LIN {X 0,Y 336.129,Z 1041.113,A -85,B 0,C 180,E1 25405.628,E2 25405.628} C_VEL
LIN {X 0,Y 318.672,Z 1080.117,A -85,B 0,C 180,E1 25408.835,E2 25408.835} C_VEL
LIN {X 0,Y 298.795,Z 1116.073,A -85,B 0,C 180,E1 25413.198,E2 25413.198} C_VEL
LIN {X 0,Y 277.626,Z 1148.443,A -85,B 0,C 180,E1 25419.027,E2 25419.027} C_VEL
LIN {X 0,Y 257.542,Z 1176.137,A -85,B 0,C 180,E1 25426.627,E2 25426.627} C_VEL
LIN {X 0,Y 241.568,Z 1197.526,A -85,B 0,C 180,E1 25435.629,E2 25435.629} C_VEL
LIN {X 0,Y 230.931,Z 1212.917,A -85,B 0,C 180,E1 25445.788,E2 25445.788} C_VEL
LIN {X 0,Y 226.21,Z 1222.177,A -85,B 0,C 180,E1 25455.992,E2 25455.992} C_VEL
LIN {X 0,Y 224.98,Z 1226.535,A -85,B 0,C 180,E1 25466.138,E2 25466.138} C_VEL
LIN {X 0,Y 225.27,Z 1226.905,A -85,B 0,C 180,E1 25470,E2 25470} C_VEL
LIN {X 0,Y 225.086,Z 1225.472,A -85,B 0,C 180,E1 25477.737,E2 25477.737} C_VEL
LIN {X 0,Y 227.29,Z 1219.666,A -85,B 0,C 180,E1 25487.457,E2 25487.457} C_VEL
LIN {X 0,Y 234.034,Z 1208.265,A -85,B 0,C 180,E1 25497.865,E2 25497.865} C_VEL
LIN {X 0,Y 246.932,Z 1190.434,A -85,B 0,C 180,E1 25507.853,E2 25507.853} C_VEL
LIN {X 0,Y 265.132,Z 1166.006,A -85,B 0,C 180,E1 25516.595,E2 25516.595} C_VEL
LIN {X 0,Y 285.468,Z 1137.166,A -85,B 0,C 180,E1 25523.324,E2 25523.324} C_VEL
LIN {X 0,Y 306.843,Z 1102.563,A -85,B 0,C 180,E1 25528.679,E2 25528.679} C_VEL
LIN {X 0,Y 326.303,Z 1064.734,A -85,B 0,C 180,E1 25532.594,E2 25532.594} C_VEL
LIN {X 0,Y 336.503,Z 1040.269,A -85,B 0,C 180,E1 25534.514,E2 25534.514} C_VEL
LIN {X 0,Y 333.813,Z 1018.325,A -85,B 0,C 180,E1 25539.751,E2 25539.751} C_VEL
LIN {X 0,Y 329.876,Z 1000.5,A -85,B 0,C 180,E1 25545.365,E2 25545.365} C_VEL
LIN {X 0,Y 326.385,Z 988.649,A -85,B 0,C 180,E1 25550.647,E2 25550.647} C_VEL
LIN {X 0,Y 324.003,Z 980.521,A -85,B 0,C 180,E1 25556.143,E2 25556.143} C_VEL
LIN {X 0,Y 323.437,Z 975.758,A -85,B 0,C 180,E1 25561.338,E2 25561.338} C_VEL
LIN {X 0,Y 323.425,Z 976.928,A -85,B 0,C 180,E1 25565.372,E2 25565.372} C_VEL
LIN {X 0,Y 325.459,Z 983.529,A -85,B 0,C 180,E1 25571.883,E2 25571.883} C_VEL
LIN {X 0,Y 329.595,Z 994.792,A -85,B 0,C 180,E1 25578.07,E2 25578.07} C_VEL
LIN {X 0,Y 334.739,Z 1011.693,A -85,B 0,C 180,E1 25584.032,E2 25584.032} C_VEL
LIN {X 0,Y 339.138,Z 1032.622,A -85,B 0,C 180,E1 25589.426,E2 25589.426} C_VEL
LIN {X 0,Y 339.403,Z 1039.091,A -85,B 0,C 180,E1 25590.675,E2 25590.675} C_VEL
LIN {X 0,Y 333.764,Z 1052.968,A -85,B 0,C 180,E1 25591.555,E2 25591.555} C_VEL
LIN {X 0,Y 325.121,Z 1067.998,A -85,B 0,C 180,E1 25592.055,E2 25592.055} C_VEL
LIN {X 0,Y 315.788,Z 1082.353,A -85,B 0,C 180,E1 25592.714,E2 25592.714} C_VEL
LIN {X 0,Y 295.451,Z 1116.69,A -85,B 0,C 180,E1 25596.74,E2 25596.74} C_VEL
LIN {X 0,Y 274.846,Z 1145.734,A -85,B 0,C 180,E1 25601.903,E2 25601.903} C_VEL
LIN {X 0,Y 255.367,Z 1169.768,A -85,B 0,C 180,E1 25608.418,E2 25608.418} C_VEL
LIN {X 0,Y 237.524,Z 1190.148,A -85,B 0,C 180,E1 25617.163,E2 25617.163} C_VEL
LIN {X 0,Y 225.183,Z 1204.304,A -85,B 0,C 180,E1 25627.237,E2 25627.237} C_VEL
LIN {X 0,Y 218.796,Z 1212.593,A -85,B 0,C 180,E1 25638.009,E2 25638.009} C_VEL
LIN {X 0,Y 217.331,Z 1215.277,A -85,B 0,C 180,E1 25646.002,E2 25646.002} C_VEL
LIN {X 0,Y 217.346,Z 1215.244,A -85,B 0,C 180,E1 25653.998,E2 25653.998} C_VEL
LIN {X 0,Y 219.664,Z 1211.343,A -85,B 0,C 180,E1 25663.972,E2 25663.972} C_VEL
LIN {X 0,Y 226.955,Z 1202.026,A -85,B 0,C 180,E1 25674.593,E2 25674.593} C_VEL
LIN {X 0,Y 239.047,Z 1188.251,A -85,B 0,C 180,E1 25683.687,E2 25683.687} C_VEL
LIN {X 0,Y 255.629,Z 1169.328,A -85,B 0,C 180,E1 25691.581,E2 25691.581} C_VEL
LIN {X 0,Y 276.15,Z 1143.785,A -85,B 0,C 180,E1 25698.386,E2 25698.386} C_VEL
LIN {X 0,Y 297.513,Z 1113.138,A -85,B 0,C 180,E1 25703.646,E2 25703.646} C_VEL
LIN {X 0,Y 316.98,Z 1079.695,A -85,B 0,C 180,E1 25707.411,E2 25707.411} C_VEL
LIN {X 0,Y 334.005,Z 1042.885,A -85,B 0,C 180,E1 25710.188,E2 25710.188} C_VEL
LIN {X 0,Y 334.535,Z 1040.217,A -85,B 0,C 180,E1 25710.507,E2 25710.507} C_VEL
LIN {X 0,Y 331.211,Z 1019.932,A -85,B 0,C 180,E1 25715.696,E2 25715.696} C_VEL
LIN {X 0,Y 327.07,Z 1004.267,A -85,B 0,C 180,E1 25721.086,E2 25721.086} C_VEL
LIN {X 0,Y 323.534,Z 993.29,A -85,B 0,C 180,E1 25726.464,E2 25726.464} C_VEL
LIN {X 0,Y 321.586,Z 987.722,A -85,B 0,C 180,E1 25730.856,E2 25730.856} C_VEL
LIN {X 0,Y 320.944,Z 983.41,A -85,B 0,C 180,E1 25735.608,E2 25735.608} C_VEL
LIN {X 0,Y 320.957,Z 983.923,A -85,B 0,C 180,E1 25740.004,E2 25740.004} C_VEL
LIN {X 0,Y 322.266,Z 991.69,A -85,B 0,C 180,E1 25746.753,E2 25746.753} C_VEL
LIN {X 0,Y 325.363,Z 1003.281,A -85,B 0,C 180,E1 25752.78,E2 25752.78} C_VEL
LIN {X 0,Y 328.73,Z 1019.789,A -85,B 0,C 180,E1 25758.475,E2 25758.475} C_VEL
LIN {X 0,Y 330.979,Z 1038.496,A -85,B 0,C 180,E1 25763.34,E2 25763.34} C_VEL
LIN {X 0,Y 331.241,Z 1043.446,A -85,B 0,C 180,E1 25764.489,E2 25764.489} C_VEL
LIN {X 0,Y 314.299,Z 1080.693,A -85,B 0,C 180,E1 25767.642,E2 25767.642} C_VEL
LIN {X 0,Y 294.401,Z 1115.737,A -85,B 0,C 180,E1 25771.868,E2 25771.868} C_VEL
LIN {X 0,Y 272.508,Z 1148.223,A -85,B 0,C 180,E1 25777.703,E2 25777.703} C_VEL
LIN {X 0,Y 252.237,Z 1175.168,A -85,B 0,C 180,E1 25785.089,E2 25785.089} C_VEL
LIN {X 0,Y 234.855,Z 1197.301,A -85,B 0,C 180,E1 25794.501,E2 25794.501} C_VEL
LIN {X 0,Y 223.565,Z 1212.701,A -85,B 0,C 180,E1 25804.936,E2 25804.936} C_VEL
LIN {X 0,Y 218.869,Z 1220.981,A -85,B 0,C 180,E1 25813.922,E2 25813.922} C_VEL
LIN {X 0,Y 217.198,Z 1225.254,A -85,B 0,C 180,E1 25821.979,E2 25821.979} C_VEL
LIN {X 0,Y 217.362,Z 1226.703,A -85,B 0,C 180,E1 25829.999,E2 25829.999} C_VEL
LIN {X 0,Y 217.194,Z 1225.269,A -85,B 0,C 180,E1 25838.02,E2 25838.02} C_VEL
LIN {X 0,Y 219.606,Z 1219.459,A -85,B 0,C 180,E1 25848.089,E2 25848.089} C_VEL
LIN {X 0,Y 227.281,Z 1207.429,A -85,B 0,C 180,E1 25859.253,E2 25859.253} C_VEL
LIN {X 0,Y 241.219,Z 1189.193,A -85,B 0,C 180,E1 25869.496,E2 25869.496} C_VEL
LIN {X 0,Y 259.567,Z 1165.746,A -85,B 0,C 180,E1 25877.91,E2 25877.91} C_VEL
LIN {X 0,Y 280.555,Z 1137.014,A -85,B 0,C 180,E1 25884.636,E2 25884.636} C_VEL
LIN {X 0,Y 302.436,Z 1102.655,A -85,B 0,C 180,E1 25889.936,E2 25889.936} C_VEL
LIN {X 0,Y 322.305,Z 1065.017,A -85,B 0,C 180,E1 25893.804,E2 25893.804} C_VEL
LIN {X 0,Y 331.473,Z 1043.453,A -85,B 0,C 180,E1 25895.529,E2 25895.529} C_VEL
LIN {X 0,Y 329.352,Z 1022.205,A -85,B 0,C 180,E1 25900.866,E2 25900.866} C_VEL
LIN {X 0,Y 325.746,Z 1004.055,A -85,B 0,C 180,E1 25906.979,E2 25906.979} C_VEL
LIN {X 0,Y 323.126,Z 993.991,A -85,B 0,C 180,E1 25911.911,E2 25911.911} C_VEL
LIN {X 0,Y 321.841,Z 988.466,A -85,B 0,C 180,E1 25915.61,E2 25915.61} C_VEL
LIN {X 0,Y 321.245,Z 983.354,A -85,B 0,C 180,E1 25921.347,E2 25921.347} C_VEL
LIN {X 0,Y 321.208,Z 984.556,A -85,B 0,C 180,E1 25925.301,E2 25925.301} C_VEL
LIN {X 0,Y 323.21,Z 991.921,A -85,B 0,C 180,E1 25932.356,E2 25932.356} C_VEL
LIN {X 0,Y 326.909,Z 1003.008,A -85,B 0,C 180,E1 25938.224,E2 25938.224} C_VEL
LIN {X 0,Y 331.466,Z 1020.386,A -85,B 0,C 180,E1 25944.284,E2 25944.284} C_VEL
LIN {X 0,Y 334.788,Z 1040.967,A -85,B 0,C 180,E1 25949.529,E2 25949.529} C_VEL
LIN {X 0,Y 317.498,Z 1079.101,A -85,B 0,C 180,E1 25952.419,E2 25952.419} C_VEL
LIN {X 0,Y 315.788,Z 1082.353,A -85,B 0,C 180,E1 25952.714,E2 25952.714} C_VEL
LIN {X 0,Y 305.838,Z 1096.298,A -85,B 0,C 180,E1 25953.5,E2 25953.5} C_VEL
LIN {X 0,Y 295.657,Z 1109.492,A -85,B 0,C 180,E1 25954.46,E2 25954.46} C_VEL
LIN {X 0,Y 275.018,Z 1138.959,A -85,B 0,C 180,E1 25959.196,E2 25959.196} C_VEL
LIN {X 0,Y 254.976,Z 1163.672,A -85,B 0,C 180,E1 25965.197,E2 25965.197} C_VEL
LIN {X 0,Y 235.982,Z 1184.766,A -85,B 0,C 180,E1 25973.177,E2 25973.177} C_VEL
LIN {X 0,Y 221.688,Z 1200.233,A -85,B 0,C 180,E1 25982.654,E2 25982.654} C_VEL
LIN {X 0,Y 212.851,Z 1210.407,A -85,B 0,C 180,E1 25993.456,E2 25993.456} C_VEL
LIN {X 0,Y 209.89,Z 1214.484,A -85,B 0,C 180,E1 26001.699,E2 26001.699} C_VEL
LIN {X 0,Y 209.529,Z 1215.793,A -85,B 0,C 180,E1 26010.001,E2 26010.001} C_VEL
LIN {X 0,Y 209.925,Z 1214.421,A -85,B 0,C 180,E1 26018.301,E2 26018.301} C_VEL
LIN {X 0,Y 214.055,Z 1208.79,A -85,B 0,C 180,E1 26028.576,E2 26028.576} C_VEL
LIN {X 0,Y 224.162,Z 1197.308,A -85,B 0,C 180,E1 26039.347,E2 26039.347} C_VEL
LIN {X 0,Y 239.611,Z 1180.675,A -85,B 0,C 180,E1 26048.524,E2 26048.524} C_VEL
LIN {X 0,Y 258.431,Z 1159.363,A -85,B 0,C 180,E1 26055.913,E2 26055.913} C_VEL
LIN {X 0,Y 279.416,Z 1132.799,A -85,B 0,C 180,E1 26061.846,E2 26061.846} C_VEL
LIN {X 0,Y 300.375,Z 1101.648,A -85,B 0,C 180,E1 26066.403,E2 26066.403} C_VEL
LIN {X 0,Y 319.816,Z 1066.366,A -85,B 0,C 180,E1 26069.79,E2 26069.79} C_VEL
LIN {X 0,Y 329.382,Z 1045.22,A -85,B 0,C 180,E1 26071.277,E2 26071.277} C_VEL
LIN {X 0,Y 327.702,Z 1028.663,A -85,B 0,C 180,E1 26075.419,E2 26075.419} C_VEL
LIN {X 0,Y 324.087,Z 1012.395,A -85,B 0,C 180,E1 26080.905,E2 26080.905} C_VEL
LIN {X 0,Y 320.969,Z 1001.103,A -85,B 0,C 180,E1 26086.354,E2 26086.354} C_VEL
LIN {X 0,Y 318.634,Z 994,A -85,B 0,C 180,E1 26092.266,E2 26092.266} C_VEL
LIN {X 0,Y 318.522,Z 991.648,A -85,B 0,C 180,E1 26094.546,E2 26094.546} C_VEL
LIN {X 0,Y 318.408,Z 990.765,A -85,B 0,C 180,E1 26097.998,E2 26097.998} C_VEL
LIN {X 0,Y 318.475,Z 994.436,A -85,B 0,C 180,E1 26102.73,E2 26102.73} C_VEL
LIN {X 0,Y 320.121,Z 1001.506,A -85,B 0,C 180,E1 26108.165,E2 26108.165} C_VEL
LIN {X 0,Y 322.618,Z 1013.068,A -85,B 0,C 180,E1 26113.582,E2 26113.582} C_VEL
LIN {X 0,Y 325.288,Z 1030.677,A -85,B 0,C 180,E1 26119.383,E2 26119.383} C_VEL
LIN {X 0,Y 326.307,Z 1047.052,A -85,B 0,C 180,E1 26123.536,E2 26123.536} C_VEL
LIN {X 0,Y 308.238,Z 1084.679,A -85,B 0,C 180,E1 26126.777,E2 26126.777} C_VEL
LIN {X 0,Y 288.882,Z 1117.376,A -85,B 0,C 180,E1 26130.803,E2 26130.803} C_VEL
LIN {X 0,Y 266.527,Z 1149.316,A -85,B 0,C 180,E1 26136.636,E2 26136.636} C_VEL
LIN {X 0,Y 245.522,Z 1176.073,A -85,B 0,C 180,E1 26144.154,E2 26144.154} C_VEL
LIN {X 0,Y 228.254,Z 1197.076,A -85,B 0,C 180,E1 26153.31,E2 26153.31} C_VEL
LIN {X 0,Y 216.224,Z 1212.484,A -85,B 0,C 180,E1 26164.023,E2 26164.023} C_VEL
LIN {X 0,Y 211.13,Z 1220.774,A -85,B 0,C 180,E1 26173.316,E2 26173.316} C_VEL
LIN {X 0,Y 209.317,Z 1225.051,A -85,B 0,C 180,E1 26181.675,E2 26181.675} C_VEL
LIN {X 0,Y 209.481,Z 1226.501,A -85,B 0,C 180,E1 26189.999,E2 26189.999} C_VEL
LIN {X 0,Y 209.313,Z 1225.066,A -85,B 0,C 180,E1 26198.324,E2 26198.324} C_VEL
LIN {X 0,Y 211.942,Z 1219.25,A -85,B 0,C 180,E1 26208.767,E2 26208.767} C_VEL
LIN {X 0,Y 220.207,Z 1207.21,A -85,B 0,C 180,E1 26220.29,E2 26220.29} C_VEL
LIN {X 0,Y 234.167,Z 1189.966,A -85,B 0,C 180,E1 26230.323,E2 26230.323} C_VEL
LIN {X 0,Y 253.486,Z 1166.351,A -85,B 0,C 180,E1 26239.037,E2 26239.037} C_VEL
LIN {X 0,Y 275.739,Z 1136.968,A -85,B 0,C 180,E1 26245.97,E2 26245.97} C_VEL
LIN {X 0,Y 297.454,Z 1103.986,A -85,B 0,C 180,E1 26251.079,E2 26251.079} C_VEL
LIN {X 0,Y 318.328,Z 1065.581,A -85,B 0,C 180,E1 26255.021,E2 26255.021} C_VEL
LIN {X 0,Y 326.534,Z 1047.208,A -85,B 0,C 180,E1 26256.454,E2 26256.454} C_VEL
LIN {X 0,Y 325.09,Z 1027.312,A -85,B 0,C 180,E1 26261.663,E2 26261.663} C_VEL
LIN {X 0,Y 322.454,Z 1011.064,A -85,B 0,C 180,E1 26267.276,E2 26267.276} C_VEL
LIN {X 0,Y 319.842,Z 999.723,A -85,B 0,C 180,E1 26273.196,E2 26273.196} C_VEL
LIN {X 0,Y 318.618,Z 992.097,A -85,B 0,C 180,E1 26279.996,E2 26279.996} C_VEL
LIN {X 0,Y 318.784,Z 990.88,A -85,B 0,C 180,E1 26283.441,E2 26283.441} C_VEL
LIN {X 0,Y 320.263,Z 998.441,A -85,B 0,C 180,E1 26291.593,E2 26291.593} C_VEL
LIN {X 0,Y 323.414,Z 1009.315,A -85,B 0,C 180,E1 26297.62,E2 26297.62} C_VEL
LIN {X 0,Y 327.03,Z 1024.806,A -85,B 0,C 180,E1 26303.247,E2 26303.247} C_VEL
LIN {X 0,Y 329.876,Z 1044.501,A -85,B 0,C 180,E1 26308.545,E2 26308.545} C_VEL
LIN {X 0,Y 311.348,Z 1083.16,A -85,B 0,C 180,E1 26311.529,E2 26311.529} C_VEL
LIN {X 0,Y 295.657,Z 1109.492,A -85,B 0,C 180,E1 26314.46,E2 26314.46} C_VEL
LIN {X 0,Y 284.954,Z 1122.218,A -85,B 0,C 180,E1 26315.603,E2 26315.603} C_VEL
LIN {X 0,Y 273.974,Z 1134.186,A -85,B 0,C 180,E1 26316.916,E2 26316.916} C_VEL
LIN {X 0,Y 251.734,Z 1161.278,A -85,B 0,C 180,E1 26323.126,E2 26323.126} C_VEL
LIN {X 0,Y 230.771,Z 1183.83,A -85,B 0,C 180,E1 26331.41,E2 26331.41} C_VEL
LIN {X 0,Y 215.941,Z 1199.01,A -85,B 0,C 180,E1 26340.581,E2 26340.581} C_VEL
LIN {X 0,Y 206.465,Z 1209.108,A -85,B 0,C 180,E1 26350.716,E2 26350.716} C_VEL
LIN {X 0,Y 202.038,Z 1214.687,A -85,B 0,C 180,E1 26361.374,E2 26361.374} C_VEL
LIN {X 0,Y 201.626,Z 1215.995,A -85,B 0,C 180,E1 26370.001,E2 26370.001} C_VEL
LIN {X 0,Y 202.075,Z 1214.625,A -85,B 0,C 180,E1 26378.626,E2 26378.626} C_VEL
LIN {X 0,Y 206.514,Z 1208.995,A -85,B 0,C 180,E1 26389.281,E2 26389.281} C_VEL
LIN {X 0,Y 217.22,Z 1197.521,A -85,B 0,C 180,E1 26400.382,E2 26400.382} C_VEL
LIN {X 0,Y 232.708,Z 1181.637,A -85,B 0,C 180,E1 26409.423,E2 26409.423} C_VEL
LIN {X 0,Y 252.937,Z 1159.61,A -85,B 0,C 180,E1 26417.213,E2 26417.213} C_VEL
LIN {X 0,Y 274.585,Z 1133.094,A -85,B 0,C 180,E1 26423.148,E2 26423.148} C_VEL
LIN {X 0,Y 295.6,Z 1102.786,A -85,B 0,C 180,E1 26427.591,E2 26427.591} C_VEL
LIN {X 0,Y 315.752,Z 1067.22,A -85,B 0,C 180,E1 26430.999,E2 26430.999} C_VEL
LIN {X 0,Y 324.701,Z 1047.502,A -85,B 0,C 180,E1 26432.46,E2 26432.46} C_VEL
LIN {X 0,Y 322.407,Z 1028.337,A -85,B 0,C 180,E1 26437.924,E2 26437.924} C_VEL
LIN {X 0,Y 319.405,Z 1014.165,A -85,B 0,C 180,E1 26443.471,E2 26443.471} C_VEL
LIN {X 0,Y 316.939,Z 1004.859,A -85,B 0,C 180,E1 26448.982,E2 26448.982} C_VEL
LIN {X 0,Y 315.947,Z 999.306,A -85,B 0,C 180,E1 26454.501,E2 26454.501} C_VEL
LIN {X 0,Y 315.866,Z 998.264,A -85,B 0,C 180,E1 26457.255,E2 26457.255} C_VEL
LIN {X 0,Y 315.693,Z 1000.868,A -85,B 0,C 180,E1 26461.579,E2 26461.579} C_VEL
LIN {X 0,Y 316.698,Z 1006.973,A -85,B 0,C 180,E1 26466.872,E2 26466.872} C_VEL
LIN {X 0,Y 318.647,Z 1017.622,A -85,B 0,C 180,E1 26472.357,E2 26472.357} C_VEL
LIN {X 0,Y 320.783,Z 1034.4,A -85,B 0,C 180,E1 26478.226,E2 26478.226} C_VEL
LIN {X 0,Y 321.419,Z 1049.974,A -85,B 0,C 180,E1 26482.374,E2 26482.374} C_VEL
LIN {X 0,Y 304.374,Z 1084.784,A -85,B 0,C 180,E1 26485.467,E2 26485.467} C_VEL
LIN {X 0,Y 284.797,Z 1117.05,A -85,B 0,C 180,E1 26489.395,E2 26489.395} C_VEL
LIN {X 0,Y 261.826,Z 1148.914,A -85,B 0,C 180,E1 26495.167,E2 26495.167} C_VEL
LIN {X 0,Y 239.876,Z 1175.832,A -85,B 0,C 180,E1 26502.747,E2 26502.747} C_VEL
LIN {X 0,Y 221.747,Z 1196.85,A -85,B 0,C 180,E1 26512.047,E2 26512.047} C_VEL
LIN {X 0,Y 208.955,Z 1212.269,A -85,B 0,C 180,E1 26523.048,E2 26523.048} C_VEL
LIN {X 0,Y 202.718,Z 1221.844,A -85,B 0,C 180,E1 26534.835,E2 26534.835} C_VEL
LIN {X 0,Y 201.238,Z 1225.927,A -85,B 0,C 180,E1 26545.681,E2 26545.681} C_VEL
LIN {X 0,Y 201.571,Z 1226.299,A -85,B 0,C 180,E1 26549.999,E2 26549.999} C_VEL
LIN {X 0,Y 201.428,Z 1224.863,A -85,B 0,C 180,E1 26558.653,E2 26558.653} C_VEL
LIN {X 0,Y 204.324,Z 1219.041,A -85,B 0,C 180,E1 26569.495,E2 26569.495} C_VEL
LIN {X 0,Y 211.786,Z 1208.752,A -85,B 0,C 180,E1 26580.055,E2 26580.055} C_VEL
LIN {X 0,Y 226.801,Z 1191.069,A -85,B 0,C 180,E1 26591.005,E2 26591.005} C_VEL
LIN {X 0,Y 247.35,Z 1167.089,A -85,B 0,C 180,E1 26600.164,E2 26600.164} C_VEL
LIN {X 0,Y 270.437,Z 1137.795,A -85,B 0,C 180,E1 26607.189,E2 26607.189} C_VEL
LIN {X 0,Y 293.829,Z 1103.238,A -85,B 0,C 180,E1 26612.515,E2 26612.515} C_VEL
LIN {X 0,Y 315.107,Z 1064.844,A -85,B 0,C 180,E1 26616.374,E2 26616.374} C_VEL
LIN {X 0,Y 321.659,Z 1050.019,A -85,B 0,C 180,E1 26617.639,E2 26617.639} C_VEL
LIN {X 0,Y 320.621,Z 1031.262,A -85,B 0,C 180,E1 26622.82,E2 26622.82} C_VEL
LIN {X 0,Y 318.609,Z 1016.255,A -85,B 0,C 180,E1 26628.338,E2 26628.338} C_VEL
LIN {X 0,Y 316.526,Z 1005.38,A -85,B 0,C 180,E1 26634.503,E2 26634.503} C_VEL
LIN {X 0,Y 316.039,Z 999.669,A -85,B 0,C 180,E1 26639.996,E2 26639.996} C_VEL
LIN {X 0,Y 316.232,Z 998.307,A -85,B 0,C 180,E1 26642.742,E2 26642.742} C_VEL
LIN {X 0,Y 317.243,Z 1005.146,A -85,B 0,C 180,E1 26651.008,E2 26651.008} C_VEL
LIN {X 0,Y 320.028,Z 1015.937,A -85,B 0,C 180,E1 26657.153,E2 26657.153} C_VEL
LIN {X 0,Y 323.16,Z 1032.088,A -85,B 0,C 180,E1 26663.112,E2 26663.112} C_VEL
LIN {X 0,Y 324.773,Z 1048.385,A -85,B 0,C 180,E1 26667.566,E2 26667.566} C_VEL
LIN {X 0,Y 306.392,Z 1085.083,A -85,B 0,C 180,E1 26670.415,E2 26670.415} C_VEL
LIN {X 0,Y 286.229,Z 1117.301,A -85,B 0,C 180,E1 26674.19,E2 26674.19} C_VEL
LIN {X 0,Y 273.974,Z 1134.186,A -85,B 0,C 180,E1 26676.916,E2 26676.916} C_VEL
LIN {X 0,Y 262.741,Z 1145.577,A -85,B 0,C 180,E1 26678.46,E2 26678.46} C_VEL
LIN {X 0,Y 251.251,Z 1156.035,A -85,B 0,C 180,E1 26680.268,E2 26680.268} C_VEL
LIN {X 0,Y 230.247,Z 1178.335,A -85,B 0,C 180,E1 26687.58,E2 26687.58} C_VEL
LIN {X 0,Y 211.68,Z 1196.622,A -85,B 0,C 180,E1 26697.529,E2 26697.529} C_VEL
LIN {X 0,Y 200.503,Z 1207.71,A -85,B 0,C 180,E1 26707.799,E2 26707.799} C_VEL
LIN {X 0,Y 195.548,Z 1213.204,A -85,B 0,C 180,E1 26716.558,E2 26716.558} C_VEL
LIN {X 0,Y 193.658,Z 1215.883,A -85,B 0,C 180,E1 26725.513,E2 26725.513} C_VEL
LIN {X 0,Y 193.675,Z 1215.852,A -85,B 0,C 180,E1 26734.488,E2 26734.488} C_VEL
LIN {X 0,Y 196.834,Z 1211.626,A -85,B 0,C 180,E1 26746.284,E2 26746.284} C_VEL
LIN {X 0,Y 206.367,Z 1201.697,A -85,B 0,C 180,E1 26758.262,E2 26758.262} C_VEL
LIN {X 0,Y 221.163,Z 1187.222,A -85,B 0,C 180,E1 26768.071,E2 26768.071} C_VEL
LIN {X 0,Y 240.486,Z 1167.55,A -85,B 0,C 180,E1 26776.235,E2 26776.235} C_VEL
LIN {X 0,Y 262.347,Z 1142.803,A -85,B 0,C 180,E1 26782.683,E2 26782.683} C_VEL
LIN {X 0,Y 284.74,Z 1113.121,A -85,B 0,C 180,E1 26787.653,E2 26787.653} C_VEL
LIN {X 0,Y 305.613,Z 1079.658,A -85,B 0,C 180,E1 26791.281,E2 26791.281} C_VEL
LIN {X 0,Y 319.634,Z 1051.823,A -85,B 0,C 180,E1 26793.391,E2 26793.391} C_VEL
LIN {X 0,Y 318.423,Z 1035.74,A -85,B 0,C 180,E1 26798.001,E2 26798.001} C_VEL
LIN {X 0,Y 316.015,Z 1021.563,A -85,B 0,C 180,E1 26803.538,E2 26803.538} C_VEL
LIN {X 0,Y 314.001,Z 1012.56,A -85,B 0,C 180,E1 26808.877,E2 26808.877} C_VEL
LIN {X 0,Y 313.072,Z 1006.838,A -85,B 0,C 180,E1 26814.45,E2 26814.45} C_VEL
LIN {X 0,Y 313.069,Z 1005.659,A -85,B 0,C 180,E1 26817.23,E2 26817.23} C_VEL
LIN {X 0,Y 312.792,Z 1008.127,A -85,B 0,C 180,E1 26821.391,E2 26821.391} C_VEL
LIN {X 0,Y 313.663,Z 1014.585,A -85,B 0,C 180,E1 26826.939,E2 26826.939} C_VEL
LIN {X 0,Y 315.164,Z 1025.492,A -85,B 0,C 180,E1 26832.438,E2 26832.438} C_VEL
LIN {X 0,Y 316.521,Z 1041.48,A -85,B 0,C 180,E1 26838.032,E2 26838.032} C_VEL
LIN {X 0,Y 316.646,Z 1053.635,A -85,B 0,C 180,E1 26841.364,E2 26841.364} C_VEL
LIN {X 0,Y 296.484,Z 1092.251,A -85,B 0,C 180,E1 26844.88,E2 26844.88} C_VEL
LIN {X 0,Y 274.08,Z 1126.511,A -85,B 0,C 180,E1 26849.451,E2 26849.451} C_VEL
LIN {X 0,Y 249.598,Z 1157.969,A -85,B 0,C 180,E1 26855.924,E2 26855.924} C_VEL
LIN {X 0,Y 227.45,Z 1183.371,A -85,B 0,C 180,E1 26864.276,E2 26864.276} C_VEL
LIN {X 0,Y 209.584,Z 1202.961,A -85,B 0,C 180,E1 26874.661,E2 26874.661} C_VEL
LIN {X 0,Y 198.615,Z 1216.095,A -85,B 0,C 180,E1 26886.259,E2 26886.259} C_VEL
LIN {X 0,Y 194.416,Z 1222.859,A -85,B 0,C 180,E1 26896.477,E2 26896.477} C_VEL
LIN {X 0,Y 193.324,Z 1225.724,A -85,B 0,C 180,E1 26905.504,E2 26905.504} C_VEL
LIN {X 0,Y 193.672,Z 1226.098,A -85,B 0,C 180,E1 26909.999,E2 26909.999} C_VEL
LIN {X 0,Y 193.548,Z 1224.66,A -85,B 0,C 180,E1 26919.008,E2 26919.008} C_VEL
LIN {X 0,Y 196.709,Z 1218.832,A -85,B 0,C 180,E1 26930.282,E2 26930.282} C_VEL
LIN {X 0,Y 204.767,Z 1208.539,A -85,B 0,C 180,E1 26941.198,E2 26941.198} C_VEL
LIN {X 0,Y 220.995,Z 1190.545,A -85,B 0,C 180,E1 26952.55,E2 26952.55} C_VEL
LIN {X 0,Y 242.803,Z 1166.166,A -85,B 0,C 180,E1 26961.855,E2 26961.855} C_VEL
LIN {X 0,Y 266.116,Z 1137.509,A -85,B 0,C 180,E1 26968.661,E2 26968.661} C_VEL
LIN {X 0,Y 290.005,Z 1103.144,A -85,B 0,C 180,E1 26973.903,E2 26973.903} C_VEL
LIN {X 0,Y 311.33,Z 1065.643,A -85,B 0,C 180,E1 26977.631,E2 26977.631} C_VEL
LIN {X 0,Y 316.873,Z 1053.738,A -85,B 0,C 180,E1 26978.641,E2 26978.641} C_VEL
LIN {X 0,Y 316.387,Z 1036.568,A -85,B 0,C 180,E1 26983.571,E2 26983.571} C_VEL
LIN {X 0,Y 314.973,Z 1022.564,A -85,B 0,C 180,E1 26988.904,E2 26988.904} C_VEL
LIN {X 0,Y 313.577,Z 1012.963,A -85,B 0,C 180,E1 26994.452,E2 26994.452} C_VEL
LIN {X 0,Y 313.14,Z 1007.127,A -85,B 0,C 180,E1 26999.996,E2 26999.996} C_VEL
LIN {X 0,Y 313.423,Z 1005.728,A -85,B 0,C 180,E1 27002.767,E2 27002.767} C_VEL
LIN {X 0,Y 314.321,Z 1012.803,A -85,B 0,C 180,E1 27011.111,E2 27011.111} C_VEL
LIN {X 0,Y 316.652,Z 1023.94,A -85,B 0,C 180,E1 27017.342,E2 27017.342} C_VEL
LIN {X 0,Y 319.119,Z 1039.538,A -85,B 0,C 180,E1 27023.074,E2 27023.074} C_VEL
LIN {X 0,Y 319.673,Z 1052.383,A -85,B 0,C 180,E1 27026.547,E2 27026.547} C_VEL
LIN {X 0,Y 301.017,Z 1087.977,A -85,B 0,C 180,E1 27029.368,E2 27029.368} C_VEL
LIN {X 0,Y 280.47,Z 1119.5,A -85,B 0,C 180,E1 27033.132,E2 27033.132} C_VEL
LIN {X 0,Y 258.044,Z 1148.187,A -85,B 0,C 180,E1 27038.362,E2 27038.362} C_VEL
LIN {X 0,Y 251.251,Z 1156.035,A -85,B 0,C 180,E1 27040.268,E2 27040.268} C_VEL
LIN {X 0,Y 239.656,Z 1165.845,A -85,B 0,C 180,E1 27042.344,E2 27042.344} C_VEL
LIN {X 0,Y 228.201,Z 1174.817,A -85,B 0,C 180,E1 27044.72,E2 27044.72} C_VEL
LIN {X 0,Y 209.305,Z 1192.808,A -85,B 0,C 180,E1 27053.599,E2 27053.599} C_VEL
LIN {X 0,Y 195.022,Z 1206.055,A -85,B 0,C 180,E1 27064.702,E2 27064.702} C_VEL
LIN {X 0,Y 187.815,Z 1213.409,A -85,B 0,C 180,E1 27075.994,E2 27075.994} C_VEL
LIN {X 0,Y 185.762,Z 1216.086,A -85,B 0,C 180,E1 27085.322,E2 27085.322} C_VEL
LIN {X 0,Y 185.779,Z 1216.055,A -85,B 0,C 180,E1 27094.679,E2 27094.679} C_VEL
LIN {X 0,Y 188.414,Z 1212.686,A -85,B 0,C 180,E1 27105.266,E2 27105.266} C_VEL
LIN {X 0,Y 197.223,Z 1203.901,A -85,B 0,C 180,E1 27117.452,E2 27117.452} C_VEL
LIN {X 0,Y 212.98,Z 1189.278,A -85,B 0,C 180,E1 27128.394,E2 27128.394} C_VEL
LIN {X 0,Y 234.289,Z 1168.566,A -85,B 0,C 180,E1 27137.391,E2 27137.391} C_VEL
LIN {X 0,Y 257.561,Z 1143.126,A -85,B 0,C 180,E1 27144.082,E2 27144.082} C_VEL
LIN {X 0,Y 280.57,Z 1113.459,A -85,B 0,C 180,E1 27149.024,E2 27149.024} C_VEL
LIN {X 0,Y 301.889,Z 1080.103,A -85,B 0,C 180,E1 27152.599,E2 27152.599} C_VEL
LIN {X 0,Y 315.02,Z 1054.626,A -85,B 0,C 180,E1 27154.586,E2 27154.586} C_VEL
LIN {X 0,Y 313.825,Z 1038.074,A -85,B 0,C 180,E1 27159.796,E2 27159.796} C_VEL
LIN {X 0,Y 311.715,Z 1024.391,A -85,B 0,C 180,E1 27165.941,E2 27165.941} C_VEL
LIN {X 0,Y 310.158,Z 1016.367,A -85,B 0,C 180,E1 27172.224,E2 27172.224} C_VEL
LIN {X 0,Y 310.197,Z 1013.042,A -85,B 0,C 180,E1 27177.205,E2 27177.205} C_VEL
LIN {X 0,Y 309.799,Z 1015.533,A -85,B 0,C 180,E1 27181.405,E2 27181.405} C_VEL
LIN {X 0,Y 310.372,Z 1022.534,A -85,B 0,C 180,E1 27187.241,E2 27187.241} C_VEL
LIN {X 0,Y 311.435,Z 1033.839,A -85,B 0,C 180,E1 27192.791,E2 27192.791} C_VEL
LIN {X 0,Y 312.074,Z 1050.249,A -85,B 0,C 180,E1 27198.397,E2 27198.397} C_VEL
LIN {X 0,Y 311.742,Z 1057.66,A -85,B 0,C 180,E1 27200.418,E2 27200.418} C_VEL
LIN {X 0,Y 291.688,Z 1094.218,A -85,B 0,C 180,E1 27203.708,E2 27203.708} C_VEL
LIN {X 0,Y 268.903,Z 1127.873,A -85,B 0,C 180,E1 27208.228,E2 27208.228} C_VEL
LIN {X 0,Y 245.167,Z 1157.406,A -85,B 0,C 180,E1 27214.295,E2 27214.295} C_VEL
LIN {X 0,Y 221.752,Z 1183.207,A -85,B 0,C 180,E1 27222.794,E2 27222.794} C_VEL
LIN {X 0,Y 202.978,Z 1202.743,A -85,B 0,C 180,E1 27233.328,E2 27233.328} C_VEL
LIN {X 0,Y 191.197,Z 1215.881,A -85,B 0,C 180,E1 27245.278,E2 27245.278} C_VEL
LIN {X 0,Y 186.174,Z 1223.299,A -85,B 0,C 180,E1 27257.566,E2 27257.566} C_VEL
LIN {X 0,Y 185.76,Z 1225.895,A -85,B 0,C 180,E1 27269.999,E2 27269.999} C_VEL
LIN {X 0,Y 186.166,Z 1223.332,A -85,B 0,C 180,E1 27282.422,E2 27282.422} C_VEL
LIN {X 0,Y 191.249,Z 1215.906,A -85,B 0,C 180,E1 27294.762,E2 27294.762} C_VEL
LIN {X 0,Y 202.964,Z 1202.834,A -85,B 0,C 180,E1 27306.674,E2 27306.674} C_VEL
LIN {X 0,Y 222.741,Z 1182.271,A -85,B 0,C 180,E1 27317.668,E2 27317.668} C_VEL
LIN {X 0,Y 246.18,Z 1156.458,A -85,B 0,C 180,E1 27325.98,E2 27325.98} C_VEL
LIN {X 0,Y 270.491,Z 1125.998,A -85,B 0,C 180,E1 27332.126,E2 27332.126} C_VEL
LIN {X 0,Y 293.906,Z 1090.969,A -85,B 0,C 180,E1 27336.687,E2 27336.687} C_VEL
LIN {X 0,Y 312.05,Z 1057.059,A -85,B 0,C 180,E1 27339.76,E2 27339.76} C_VEL
LIN {X 0,Y 312.086,Z 1040.89,A -85,B 0,C 180,E1 27344.679,E2 27344.679} C_VEL
LIN {X 0,Y 311.146,Z 1027.417,A -85,B 0,C 180,E1 27350.185,E2 27350.185} C_VEL
LIN {X 0,Y 310.173,Z 1018.56,A -85,B 0,C 180,E1 27355.795,E2 27355.795} C_VEL
LIN {X 0,Y 310.191,Z 1014.57,A -85,B 0,C 180,E1 27359.996,E2 27359.996} C_VEL
LIN {X 0,Y 310.532,Z 1013.159,A -85,B 0,C 180,E1 27362.792,E2 27362.792} C_VEL
LIN {X 0,Y 311.158,Z 1020.346,A -85,B 0,C 180,E1 27371.226,E2 27371.226} C_VEL
LIN {X 0,Y 312.94,Z 1030.439,A -85,B 0,C 180,E1 27376.881,E2 27376.881} C_VEL
LIN {X 0,Y 314.776,Z 1045.697,A -85,B 0,C 180,E1 27382.64,E2 27382.64} C_VEL
LIN {X 0,Y 315.074,Z 1055.457,A -85,B 0,C 180,E1 27385.427,E2 27385.427} C_VEL
LIN {X 0,Y 294.26,Z 1093.323,A -85,B 0,C 180,E1 27388.523,E2 27388.523} C_VEL
LIN {X 0,Y 271.971,Z 1125.572,A -85,B 0,C 180,E1 27392.61,E2 27392.61} C_VEL
LIN {X 0,Y 247.138,Z 1155.256,A -85,B 0,C 180,E1 27398.58,E2 27398.58} C_VEL
LIN {X 0,Y 228.201,Z 1174.817,A -85,B 0,C 180,E1 27404.72,E2 27404.72} C_VEL
LIN {X 0,Y 216.936,Z 1183.036,A -85,B 0,C 180,E1 27407.457,E2 27407.457} C_VEL
LIN {X 0,Y 205.955,Z 1190.377,A -85,B 0,C 180,E1 27410.58,E2 27410.58} C_VEL
LIN {X 0,Y 190.068,Z 1204.272,A -85,B 0,C 180,E1 27421.424,E2 27421.424} C_VEL
LIN {X 0,Y 181.17,Z 1212.451,A -85,B 0,C 180,E1 27432.979,E2 27432.979} C_VEL
LIN {X 0,Y 177.881,Z 1216.287,A -85,B 0,C 180,E1 27445.114,E2 27445.114} C_VEL
LIN {X 0,Y 177.898,Z 1216.258,A -85,B 0,C 180,E1 27454.887,E2 27454.887} C_VEL
LIN {X 0,Y 180.735,Z 1212.89,A -85,B 0,C 180,E1 27465.931,E2 27465.931} C_VEL
LIN {X 0,Y 190.881,Z 1203.459,A -85,B 0,C 180,E1 27479.205,E2 27479.205} C_VEL
LIN {X 0,Y 206.787,Z 1189.499,A -85,B 0,C 180,E1 27489.767,E2 27489.767} C_VEL
LIN {X 0,Y 227.992,Z 1169.808,A -85,B 0,C 180,E1 27498.527,E2 27498.527} C_VEL
LIN {X 0,Y 251.718,Z 1144.892,A -85,B 0,C 180,E1 27505.24,E2 27505.24} C_VEL
LIN {X 0,Y 276.474,Z 1113.939,A -85,B 0,C 180,E1 27510.414,E2 27510.414} C_VEL
LIN {X 0,Y 299.094,Z 1079.171,A -85,B 0,C 180,E1 27514.062,E2 27514.062} C_VEL
LIN {X 0,Y 310.204,Z 1057.933,A -85,B 0,C 180,E1 27515.778,E2 27515.778} C_VEL
LIN {X 0,Y 309.459,Z 1041.591,A -85,B 0,C 180,E1 27521.307,E2 27521.307} C_VEL
LIN {X 0,Y 307.962,Z 1029.714,A -85,B 0,C 180,E1 27527.169,E2 27527.169} C_VEL
LIN {X 0,Y 306.921,Z 1021.705,A -85,B 0,C 180,E1 27534.339,E2 27534.339} C_VEL
LIN {X 0,Y 307.027,Z 1020.327,A -85,B 0,C 180,E1 27537.176,E2 27537.176} C_VEL
LIN {X 0,Y 306.569,Z 1022.834,A -85,B 0,C 180,E1 27541.42,E2 27541.42} C_VEL
LIN {X 0,Y 306.897,Z 1030.059,A -85,B 0,C 180,E1 27547.323,E2 27547.323} C_VEL
LIN {X 0,Y 307.513,Z 1041.42,A -85,B 0,C 180,E1 27552.827,E2 27552.827} C_VEL
LIN {X 0,Y 307.317,Z 1058.006,A -85,B 0,C 180,E1 27558.464,E2 27558.464} C_VEL
LIN {X 0,Y 307.006,Z 1061.117,A -85,B 0,C 180,E1 27559.304,E2 27559.304} C_VEL
LIN {X 0,Y 286.252,Z 1097.354,A -85,B 0,C 180,E1 27562.62,E2 27562.62} C_VEL
LIN {X 0,Y 264.171,Z 1128.814,A -85,B 0,C 180,E1 27566.891,E2 27566.891} C_VEL
LIN {X 0,Y 240.263,Z 1157.566,A -85,B 0,C 180,E1 27572.797,E2 27572.797} C_VEL
LIN {X 0,Y 216.562,Z 1182.701,A -85,B 0,C 180,E1 27581.081,E2 27581.081} C_VEL
LIN {X 0,Y 196.492,Z 1202.525,A -85,B 0,C 180,E1 27591.906,E2 27591.906} C_VEL
LIN {X 0,Y 184.607,Z 1214.77,A -85,B 0,C 180,E1 27603.162,E2 27603.162} C_VEL
LIN {X 0,Y 178.844,Z 1222.448,A -85,B 0,C 180,E1 27615.274,E2 27615.274} C_VEL
LIN {X 0,Y 177.501,Z 1225.318,A -85,B 0,C 180,E1 27625.102,E2 27625.102} C_VEL
LIN {X 0,Y 177.847,Z 1225.693,A -85,B 0,C 180,E1 27629.999,E2 27629.999} C_VEL
LIN {X 0,Y 177.833,Z 1224.254,A -85,B 0,C 180,E1 27639.811,E2 27639.811} C_VEL
LIN {X 0,Y 181.624,Z 1218.432,A -85,B 0,C 180,E1 27652.025,E2 27652.025} C_VEL
LIN {X 0,Y 192.25,Z 1206.782,A -85,B 0,C 180,E1 27664.85,E2 27664.85} C_VEL
LIN {X 0,Y 210.292,Z 1189.037,A -85,B 0,C 180,E1 27676.1,E2 27676.1} C_VEL
LIN {X 0,Y 232.935,Z 1165.81,A -85,B 0,C 180,E1 27684.968,E2 27684.968} C_VEL
LIN {X 0,Y 258.008,Z 1136.921,A -85,B 0,C 180,E1 27691.757,E2 27691.757} C_VEL
LIN {X 0,Y 282.494,Z 1103.567,A -85,B 0,C 180,E1 27696.718,E2 27696.718} C_VEL
LIN {X 0,Y 304.875,Z 1065.952,A -85,B 0,C 180,E1 27700.341,E2 27700.341} C_VEL
LIN {X 0,Y 307.088,Z 1061.552,A -85,B 0,C 180,E1 27700.67,E2 27700.67} C_VEL
LIN {X 0,Y 307.75,Z 1047.361,A -85,B 0,C 180,E1 27705.019,E2 27705.019} C_VEL
LIN {X 0,Y 307.33,Z 1033.767,A -85,B 0,C 180,E1 27710.707,E2 27710.707} C_VEL
LIN {X 0,Y 306.793,Z 1024.468,A -85,B 0,C 180,E1 27717.166,E2 27717.166} C_VEL
LIN {X 0,Y 307.343,Z 1020.474,A -85,B 0,C 180,E1 27722.821,E2 27722.821} C_VEL
LIN {X 0,Y 307.904,Z 1027.849,A -85,B 0,C 180,E1 27731.346,E2 27731.346} C_VEL
LIN {X 0,Y 309.215,Z 1038.271,A -85,B 0,C 180,E1 27737.091,E2 27737.091} C_VEL
LIN {X 0,Y 310.336,Z 1053.068,A -85,B 0,C 180,E1 27742.603,E2 27742.603} C_VEL
LIN {X 0,Y 310.383,Z 1058.259,A -85,B 0,C 180,E1 27744.169,E2 27744.169} C_VEL
LIN {X 0,Y 289.812,Z 1094.82,A -85,B 0,C 180,E1 27747.272,E2 27747.272} C_VEL
LIN {X 0,Y 266.424,Z 1127.522,A -85,B 0,C 180,E1 27751.447,E2 27751.447} C_VEL
LIN {X 0,Y 242.239,Z 1155.5,A -85,B 0,C 180,E1 27757.103,E2 27757.103} C_VEL
LIN {X 0,Y 218.71,Z 1178.774,A -85,B 0,C 180,E1 27764.753,E2 27764.753} C_VEL
LIN {X 0,Y 205.955,Z 1190.377,A -85,B 0,C 180,E1 27770.58,E2 27770.58} C_VEL
LIN {X 0,Y 195.419,Z 1196.861,A -85,B 0,C 180,E1 27774.136,E2 27774.136} C_VEL
LIN {X 0,Y 185.534,Z 1202.435,A -85,B 0,C 180,E1 27778.164,E2 27778.164} C_VEL
LIN {X 0,Y 175.021,Z 1211.434,A -85,B 0,C 180,E1 27789.739,E2 27789.739} C_VEL
LIN {X 0,Y 170.713,Z 1215.5,A -85,B 0,C 180,E1 27799.775,E2 27799.775} C_VEL
LIN {X 0,Y 170.035,Z 1216.802,A -85,B 0,C 180,E1 27810.001,E2 27810.001} C_VEL
LIN {X 0,Y 172.261,Z 1213.978,A -85,B 0,C 180,E1 27824.707,E2 27824.707} C_VEL
LIN {X 0,Y 181.945,Z 1205.403,A -85,B 0,C 180,E1 27838.613,E2 27838.613} C_VEL
LIN {X 0,Y 199.375,Z 1190.879,A -85,B 0,C 180,E1 27850.561,E2 27850.561} C_VEL
LIN {X 0,Y 221.521,Z 1171.242,A -85,B 0,C 180,E1 27859.647,E2 27859.647} C_VEL
LIN {X 0,Y 247.243,Z 1145.196,A -85,B 0,C 180,E1 27866.747,E2 27866.747} C_VEL
LIN {X 0,Y 271.86,Z 1115.362,A -85,B 0,C 180,E1 27871.724,E2 27871.724} C_VEL
LIN {X 0,Y 294.945,Z 1080.975,A -85,B 0,C 180,E1 27875.328,E2 27875.328} C_VEL
LIN {X 0,Y 304.967,Z 1062.934,A -85,B 0,C 180,E1 27876.683,E2 27876.683} C_VEL
LIN {X 0,Y 305.386,Z 1052.105,A -85,B 0,C 180,E1 27880.109,E2 27880.109} C_VEL
LIN {X 0,Y 304.592,Z 1039.665,A -85,B 0,C 180,E1 27885.605,E2 27885.605} C_VEL
LIN {X 0,Y 303.657,Z 1031.621,A -85,B 0,C 180,E1 27891.396,E2 27891.396} C_VEL
LIN {X 0,Y 303.817,Z 1027.586,A -85,B 0,C 180,E1 27897.146,E2 27897.146} C_VEL
LIN {X 0,Y 303.192,Z 1030.314,A -85,B 0,C 180,E1 27901.686,E2 27901.686} C_VEL
LIN {X 0,Y 303.284,Z 1038.497,A -85,B 0,C 180,E1 27908.016,E2 27908.016} C_VEL
LIN {X 0,Y 303.249,Z 1051.147,A -85,B 0,C 180,E1 27913.731,E2 27913.731} C_VEL
LIN {X 0,Y 302.502,Z 1064.102,A -85,B 0,C 180,E1 27918.054,E2 27918.054} C_VEL
LIN {X 0,Y 280.922,Z 1100.49,A -85,B 0,C 180,E1 27921.492,E2 27921.492} C_VEL
LIN {X 0,Y 258.184,Z 1131.456,A -85,B 0,C 180,E1 27925.781,E2 27925.781} C_VEL
LIN {X 0,Y 233.778,Z 1159.547,A -85,B 0,C 180,E1 27931.728,E2 27931.728} C_VEL
LIN {X 0,Y 209.789,Z 1183.837,A -85,B 0,C 180,E1 27940.021,E2 27940.021} C_VEL
LIN {X 0,Y 190.139,Z 1202.306,A -85,B 0,C 180,E1 27950.39,E2 27950.39} C_VEL
LIN {X 0,Y 175.628,Z 1216.512,A -85,B 0,C 180,E1 27964.443,E2 27964.443} C_VEL
LIN {X 0,Y 170.143,Z 1223.588,A -85,B 0,C 180,E1 27978.385,E2 27978.385} C_VEL
LIN {X 0,Y 169.933,Z 1225.491,A -85,B 0,C 180,E1 27989.999,E2 27989.999} C_VEL
LIN {X 0,Y 170.154,Z 1223.611,A -85,B 0,C 180,E1 28001.633,E2 28001.633} C_VEL
LIN {X 0,Y 175.66,Z 1216.565,A -85,B 0,C 180,E1 28015.55,E2 28015.55} C_VEL
LIN {X 0,Y 190.131,Z 1202.404,A -85,B 0,C 180,E1 28029.611,E2 28029.611} C_VEL
LIN {X 0,Y 211.274,Z 1182.545,A -85,B 0,C 180,E1 28040.636,E2 28040.636} C_VEL
LIN {X 0,Y 236.941,Z 1156.454,A -85,B 0,C 180,E1 28049.125,E2 28049.125} C_VEL
LIN {X 0,Y 262.941,Z 1125.827,A -85,B 0,C 180,E1 28055.182,E2 28055.182} C_VEL
LIN {X 0,Y 287.103,Z 1091.436,A -85,B 0,C 180,E1 28059.524,E2 28059.524} C_VEL
LIN {X 0,Y 302.708,Z 1064.094,A -85,B 0,C 180,E1 28062.007,E2 28062.007} C_VEL
LIN {X 0,Y 303.466,Z 1049.427,A -85,B 0,C 180,E1 28067.014,E2 28067.014} C_VEL
LIN {X 0,Y 303.462,Z 1038.455,A -85,B 0,C 180,E1 28072.176,E2 28072.176} C_VEL
LIN {X 0,Y 303.39,Z 1030.564,A -85,B 0,C 180,E1 28078.422,E2 28078.422} C_VEL
LIN {X 0,Y 304.118,Z 1027.758,A -85,B 0,C 180,E1 28082.851,E2 28082.851} C_VEL
LIN {X 0,Y 304.072,Z 1033.314,A -85,B 0,C 180,E1 28089.912,E2 28089.912} C_VEL
LIN {X 0,Y 305.08,Z 1042.97,A -85,B 0,C 180,E1 28095.845,E2 28095.845} C_VEL
LIN {X 0,Y 305.74,Z 1057.726,A -85,B 0,C 180,E1 28101.72,E2 28101.72} C_VEL
LIN {X 0,Y 305.228,Z 1062.974,A -85,B 0,C 180,E1 28103.21,E2 28103.21} C_VEL
LIN {X 0,Y 284.73,Z 1097.457,A -85,B 0,C 180,E1 28106.096,E2 28106.096} C_VEL
LIN {X 0,Y 262.358,Z 1127.807,A -85,B 0,C 180,E1 28109.964,E2 28109.964} C_VEL
LIN {X 0,Y 237.51,Z 1155.742,A -85,B 0,C 180,E1 28115.568,E2 28115.568} C_VEL
LIN {X 0,Y 213.041,Z 1179.081,A -85,B 0,C 180,E1 28123.26,E2 28123.26} C_VEL
LIN {X 0,Y 191.86,Z 1197.248,A -85,B 0,C 180,E1 28133.677,E2 28133.677} C_VEL
LIN {X 0,Y 185.534,Z 1202.435,A -85,B 0,C 180,E1 28138.164,E2 28138.164} C_VEL
LIN {X 0,Y 176.412,Z 1207.15,A -85,B 0,C 180,E1 28142.675,E2 28142.675} C_VEL
LIN {X 0,Y 168.266,Z 1210.987,A -85,B 0,C 180,E1 28147.688,E2 28147.688} C_VEL
LIN {X 0,Y 162.924,Z 1215.702,A -85,B 0,C 180,E1 28159.281,E2 28159.281} C_VEL
LIN {X 0,Y 162.141,Z 1217.004,A -85,B 0,C 180,E1 28170.001,E2 28170.001} C_VEL
LIN {X 0,Y 162.967,Z 1215.645,A -85,B 0,C 180,E1 28180.718,E2 28180.718} C_VEL
LIN {X 0,Y 169.386,Z 1210.022,A -85,B 0,C 180,E1 28193.739,E2 28193.739} C_VEL
LIN {X 0,Y 183.829,Z 1198.581,A -85,B 0,C 180,E1 28206.7,E2 28206.7} C_VEL
LIN {X 0,Y 203.389,Z 1182.779,A -85,B 0,C 180,E1 28216.586,E2 28216.586} C_VEL
LIN {X 0,Y 227.731,Z 1160.862,A -85,B 0,C 180,E1 28224.598,E2 28224.598} C_VEL
LIN {X 0,Y 252.745,Z 1134.563,A -85,B 0,C 180,E1 28230.381,E2 28230.381} C_VEL
LIN {X 0,Y 277.56,Z 1102.925,A -85,B 0,C 180,E1 28234.717,E2 28234.717} C_VEL
LIN {X 0,Y 300.009,Z 1067.06,A -85,B 0,C 180,E1 28237.816,E2 28237.816} C_VEL
LIN {X 0,Y 300.813,Z 1063.626,A -85,B 0,C 180,E1 28238.59,E2 28238.59} C_VEL
LIN {X 0,Y 300.783,Z 1050.23,A -85,B 0,C 180,E1 28243.921,E2 28243.921} C_VEL
LIN {X 0,Y 300.413,Z 1042.421,A -85,B 0,C 180,E1 28248.367,E2 28248.367} C_VEL
LIN {X 0,Y 300.066,Z 1036.264,A -85,B 0,C 180,E1 28254.209,E2 28254.209} C_VEL
LIN {X 0,Y 300.305,Z 1034.689,A -85,B 0,C 180,E1 28257.112,E2 28257.112} C_VEL
LIN {X 0,Y 299.55,Z 1038.642,A -85,B 0,C 180,E1 28262.903,E2 28262.903} C_VEL
LIN {X 0,Y 299.309,Z 1047.018,A -85,B 0,C 180,E1 28268.737,E2 28268.737} C_VEL
LIN {X 0,Y 298.628,Z 1059.63,A -85,B 0,C 180,E1 28274.158,E2 28274.158} C_VEL
LIN {X 0,Y 297.918,Z 1067.613,A -85,B 0,C 180,E1 28276.863,E2 28276.863} C_VEL
LIN {X 0,Y 274.915,Z 1104.724,A -85,B 0,C 180,E1 28280.443,E2 28280.443} C_VEL
LIN {X 0,Y 249.167,Z 1137.894,A -85,B 0,C 180,E1 28285.294,E2 28285.294} C_VEL
LIN {X 0,Y 223.039,Z 1166.034,A -85,B 0,C 180,E1 28291.871,E2 28291.871} C_VEL
LIN {X 0,Y 199.269,Z 1188.435,A -85,B 0,C 180,E1 28300.497,E2 28300.497} C_VEL
LIN {X 0,Y 179.102,Z 1206.25,A -85,B 0,C 180,E1 28312.164,E2 28312.164} C_VEL
LIN {X 0,Y 167.252,Z 1217.369,A -85,B 0,C 180,E1 28324.941,E2 28324.941} C_VEL
LIN {X 0,Y 162.129,Z 1223.829,A -85,B 0,C 180,E1 28339.226,E2 28339.226} C_VEL
LIN {X 0,Y 162.039,Z 1225.289,A -85,B 0,C 180,E1 28349.999,E2 28349.999} C_VEL
LIN {X 0,Y 162.129,Z 1223.847,A -85,B 0,C 180,E1 28360.773,E2 28360.773} C_VEL
LIN {X 0,Y 167.311,Z 1217.395,A -85,B 0,C 180,E1 28375.102,E2 28375.102} C_VEL
LIN {X 0,Y 179.089,Z 1206.349,A -85,B 0,C 180,E1 28387.837,E2 28387.837} C_VEL
LIN {X 0,Y 199.245,Z 1188.572,A -85,B 0,C 180,E1 28399.509,E2 28399.509} C_VEL
LIN {X 0,Y 224.392,Z 1164.894,A -85,B 0,C 180,E1 28408.489,E2 28408.489} C_VEL
LIN {X 0,Y 250.704,Z 1136.322,A -85,B 0,C 180,E1 28415.041,E2 28415.041} C_VEL
LIN {X 0,Y 276.482,Z 1102.822,A -85,B 0,C 180,E1 28419.809,E2 28419.809} C_VEL
LIN {X 0,Y 298.111,Z 1067.788,A -85,B 0,C 180,E1 28423.14,E2 28423.14} C_VEL
LIN {X 0,Y 299.312,Z 1053.575,A -85,B 0,C 180,E1 28428.316,E2 28428.316} C_VEL
LIN {X 0,Y 299.583,Z 1043.592,A -85,B 0,C 180,E1 28433.463,E2 28433.463} C_VEL
LIN {X 0,Y 300.083,Z 1036.325,A -85,B 0,C 180,E1 28439.996,E2 28439.996} C_VEL
LIN {X 0,Y 300.572,Z 1034.916,A -85,B 0,C 180,E1 28442.885,E2 28442.885} C_VEL
LIN {X 0,Y 300.487,Z 1040.815,A -85,B 0,C 180,E1 28450.159,E2 28450.159} C_VEL
LIN {X 0,Y 300.986,Z 1050.64,A -85,B 0,C 180,E1 28456.068,E2 28456.068} C_VEL
LIN {X 0,Y 300.923,Z 1065.286,A -85,B 0,C 180,E1 28461.789,E2 28461.789} C_VEL
LIN {X 0,Y 297.564,Z 1071.886,A -85,B 0,C 180,E1 28462.422,E2 28462.422} C_VEL
LIN {X 0,Y 275.132,Z 1106.694,A -85,B 0,C 180,E1 28465.598,E2 28465.598} C_VEL
LIN {X 0,Y 251.152,Z 1136.669,A -85,B 0,C 180,E1 28469.855,E2 28469.855} C_VEL
LIN {X 0,Y 225.003,Z 1163.73,A -85,B 0,C 180,E1 28476.086,E2 28476.086} C_VEL
LIN {X 0,Y 201.029,Z 1184.927,A -85,B 0,C 180,E1 28484.269,E2 28484.269} C_VEL
LIN {X 0,Y 180.54,Z 1201.342,A -85,B 0,C 180,E1 28495.492,E2 28495.492} C_VEL
LIN {X 0,Y 168.266,Z 1210.987,A -85,B 0,C 180,E1 28507.688,E2 28507.688} C_VEL
LIN {X 0,Y 165.273,Z 1212.618,A -85,B 0,C 180,E1 28510.455,E2 28510.455} C_VEL
LIN {X 0,Y 155.343,Z 1215.813,A -85,B 0,C 180,E1 28518.302,E2 28518.302} C_VEL
LIN {X 0,Y 155.021,Z 1215.971,A -85,B 0,C 180,E1 28519.104,E2 28519.104} C_VEL
LIN {X 0,Y 154.236,Z 1217.206,A -85,B 0,C 180,E1 28530.001,E2 28530.001} C_VEL
LIN {X 0,Y 155.893,Z 1215.132,A -85,B 0,C 180,E1 28543.684,E2 28543.684} C_VEL
LIN {X 0,Y 164.287,Z 1208.615,A -85,B 0,C 180,E1 28557.463,E2 28557.463} C_VEL
LIN {X 0,Y 181.141,Z 1196.134,A -85,B 0,C 180,E1 28570.415,E2 28570.415} C_VEL
LIN {X 0,Y 203.978,Z 1178.175,A -85,B 0,C 180,E1 28580.457,E2 28580.457} C_VEL
LIN {X 0,Y 230.108,Z 1154.574,A -85,B 0,C 180,E1 28587.978,E2 28587.978} C_VEL
LIN {X 0,Y 257.538,Z 1124.868,A -85,B 0,C 180,E1 28593.536,E2 28593.536} C_VEL
LIN {X 0,Y 282.23,Z 1091.805,A -85,B 0,C 180,E1 28597.339,E2 28597.339} C_VEL
LIN {X 0,Y 295.829,Z 1069.807,A -85,B 0,C 180,E1 28599.072,E2 28599.072} C_VEL
LIN {X 0,Y 296.571,Z 1057.922,A -85,B 0,C 180,E1 28603.659,E2 28603.659} C_VEL
LIN {X 0,Y 296.361,Z 1048.166,A -85,B 0,C 180,E1 28609.38,E2 28609.38} C_VEL
LIN {X 0,Y 296.407,Z 1043.45,A -85,B 0,C 180,E1 28614.137,E2 28614.137} C_VEL
LIN {X 0,Y 296.751,Z 1041.797,A -85,B 0,C 180,E1 28617.078,E2 28617.078} C_VEL
LIN {X 0,Y 295.935,Z 1044.349,A -85,B 0,C 180,E1 28621.471,E2 28621.471} C_VEL
LIN {X 0,Y 295.339,Z 1051.773,A -85,B 0,C 180,E1 28627.372,E2 28627.372} C_VEL
LIN {X 0,Y 294.374,Z 1062.685,A -85,B 0,C 180,E1 28632.561,E2 28632.561} C_VEL
LIN {X 0,Y 293.399,Z 1070.682,A -85,B 0,C 180,E1 28635.507,E2 28635.507} C_VEL
LIN {X 0,Y 290.731,Z 1075.888,A -85,B 0,C 180,E1 28636.139,E2 28636.139} C_VEL
LIN {X 0,Y 267.525,Z 1110.631,A -85,B 0,C 180,E1 28639.577,E2 28639.577} C_VEL
LIN {X 0,Y 243.194,Z 1140.439,A -85,B 0,C 180,E1 28644.101,E2 28644.101} C_VEL
LIN {X 0,Y 217.483,Z 1167.023,A -85,B 0,C 180,E1 28650.433,E2 28650.433} C_VEL
LIN {X 0,Y 191.822,Z 1190.111,A -85,B 0,C 180,E1 28659.627,E2 28659.627} C_VEL
LIN {X 0,Y 171.16,Z 1207.394,A -85,B 0,C 180,E1 28671.704,E2 28671.704} C_VEL
LIN {X 0,Y 157.847,Z 1219.324,A -85,B 0,C 180,E1 28687.418,E2 28687.418} C_VEL
LIN {X 0,Y 154.22,Z 1223.736,A -85,B 0,C 180,E1 28699.242,E2 28699.242} C_VEL
LIN {X 0,Y 154.123,Z 1225.087,A -85,B 0,C 180,E1 28709.999,E2 28709.999} C_VEL
LIN {X 0,Y 154.299,Z 1223.644,A -85,B 0,C 180,E1 28721.326,E2 28721.326} C_VEL
LIN {X 0,Y 159.725,Z 1217.445,A -85,B 0,C 180,E1 28735.907,E2 28735.907} C_VEL
LIN {X 0,Y 172.72,Z 1206.131,A -85,B 0,C 180,E1 28749.497,E2 28749.497} C_VEL
LIN {X 0,Y 194.043,Z 1188.343,A -85,B 0,C 180,E1 28761.343,E2 28761.343} C_VEL
LIN {X 0,Y 220.203,Z 1164.637,A -85,B 0,C 180,E1 28770.315,E2 28770.315} C_VEL
LIN {X 0,Y 247.381,Z 1136.024,A -85,B 0,C 180,E1 28776.75,E2 28776.75} C_VEL
LIN {X 0,Y 273.701,Z 1102.591,A -85,B 0,C 180,E1 28781.383,E2 28781.383} C_VEL
LIN {X 0,Y 293.531,Z 1071.263,A -85,B 0,C 180,E1 28784.361,E2 28784.361} C_VEL
LIN {X 0,Y 295.101,Z 1057.715,A -85,B 0,C 180,E1 28789.645,E2 28789.645} C_VEL
LIN {X 0,Y 295.641,Z 1049.73,A -85,B 0,C 180,E1 28794.114,E2 28794.114} C_VEL
LIN {X 0,Y 296.411,Z 1043.447,A -85,B 0,C 180,E1 28799.996,E2 28799.996} C_VEL
LIN {X 0,Y 296.988,Z 1042.058,A -85,B 0,C 180,E1 28802.92,E2 28802.92} C_VEL
LIN {X 0,Y 296.631,Z 1048.666,A -85,B 0,C 180,E1 28810.79,E2 28810.79} C_VEL
LIN {X 0,Y 296.737,Z 1059.091,A -85,B 0,C 180,E1 28816.684,E2 28816.684} C_VEL
LIN {X 0,Y 296.252,Z 1069.61,A -85,B 0,C 180,E1 28820.81,E2 28820.81} C_VEL
LIN {X 0,Y 273.361,Z 1104.943,A -85,B 0,C 180,E1 28823.848,E2 28823.848} C_VEL
LIN {X 0,Y 247.285,Z 1136.937,A -85,B 0,C 180,E1 28828.255,E2 28828.255} C_VEL
LIN {X 0,Y 220.394,Z 1163.963,A -85,B 0,C 180,E1 28834.408,E2 28834.408} C_VEL
LIN {X 0,Y 195.543,Z 1185.142,A -85,B 0,C 180,E1 28842.595,E2 28842.595} C_VEL
LIN {X 0,Y 174.017,Z 1201.547,A -85,B 0,C 180,E1 28854.002,E2 28854.002} C_VEL
LIN {X 0,Y 160.141,Z 1211.845,A -85,B 0,C 180,E1 28867.761,E2 28867.761} C_VEL
LIN {X 0,Y 155.021,Z 1215.971,A -85,B 0,C 180,E1 28879.104,E2 28879.104} C_VEL
LIN {X 0,Y 150.246,Z 1217.066,A -85,B 0,C 180,E1 28885.394,E2 28885.394} C_VEL
LIN {X 0,Y 146.172,Z 1217.292,A -85,B 0,C 180,E1 28892.042,E2 28892.042} C_VEL
LIN {X 0,Y 149.592,Z 1214.349,A -85,B 0,C 180,E1 28907.692,E2 28907.692} C_VEL
LIN {X 0,Y 160.047,Z 1206.828,A -85,B 0,C 180,E1 28921.598,E2 28921.598} C_VEL
LIN {X 0,Y 179.291,Z 1193.273,A -85,B 0,C 180,E1 28934.297,E2 28934.297} C_VEL
LIN {X 0,Y 202.713,Z 1175.29,A -85,B 0,C 180,E1 28943.449,E2 28943.449} C_VEL
LIN {X 0,Y 229.231,Z 1151.634,A -85,B 0,C 180,E1 28950.405,E2 28950.405} C_VEL
LIN {X 0,Y 255.818,Z 1123.095,A -85,B 0,C 180,E1 28955.418,E2 28955.418} C_VEL
LIN {X 0,Y 280.071,Z 1090.993,A -85,B 0,C 180,E1 28958.938,E2 28958.938} C_VEL
LIN {X 0,Y 291.024,Z 1073.717,A -85,B 0,C 180,E1 28960.264,E2 28960.264} C_VEL
LIN {X 0,Y 292.135,Z 1063.815,A -85,B 0,C 180,E1 28964.206,E2 28964.206} C_VEL
LIN {X 0,Y 292.399,Z 1054.495,A -85,B 0,C 180,E1 28969.944,E2 28969.944} C_VEL
LIN {X 0,Y 292.891,Z 1048.757,A -85,B 0,C 180,E1 28977.039,E2 28977.039} C_VEL
LIN {X 0,Y 291.982,Z 1051.674,A -85,B 0,C 180,E1 28981.822,E2 28981.822} C_VEL
LIN {X 0,Y 291.026,Z 1059.276,A -85,B 0,C 180,E1 28987.632,E2 28987.632} C_VEL
LIN {X 0,Y 289.487,Z 1070.518,A -85,B 0,C 180,E1 28992.808,E2 28992.808} C_VEL
LIN {X 0,Y 288.644,Z 1075.337,A -85,B 0,C 180,E1 28994.589,E2 28994.589} C_VEL
LIN {X 0,Y 265.532,Z 1109.489,A -85,B 0,C 180,E1 28997.84,E2 28997.84} C_VEL
LIN {X 0,Y 239.678,Z 1140.485,A -85,B 0,C 180,E1 29002.389,E2 29002.389} C_VEL
LIN {X 0,Y 213.471,Z 1166.778,A -85,B 0,C 180,E1 29008.546,E2 29008.546} C_VEL
LIN {X 0,Y 186.55,Z 1190.007,A -85,B 0,C 180,E1 29017.758,E2 29017.758} C_VEL
LIN {X 0,Y 164.824,Z 1207.179,A -85,B 0,C 180,E1 29029.943,E2 29029.943} C_VEL
LIN {X 0,Y 150.417,Z 1219.117,A -85,B 0,C 180,E1 29046.236,E2 29046.236} C_VEL
LIN {X 0,Y 146.465,Z 1223.421,A -85,B 0,C 180,E1 29058.058,E2 29058.058} C_VEL
LIN {X 0,Y 146.228,Z 1224.885,A -85,B 0,C 180,E1 29069.999,E2 29069.999} C_VEL
LIN {X 0,Y 146.464,Z 1223.44,A -85,B 0,C 180,E1 29081.941,E2 29081.941} C_VEL
LIN {X 0,Y 152.63,Z 1217.087,A -85,B 0,C 180,E1 29097.498,E2 29097.498} C_VEL
LIN {X 0,Y 166.492,Z 1205.916,A -85,B 0,C 180,E1 29111.287,E2 29111.287} C_VEL
LIN {X 0,Y 189.06,Z 1188.113,A -85,B 0,C 180,E1 29123.272,E2 29123.272} C_VEL
LIN {X 0,Y 216.274,Z 1164.382,A -85,B 0,C 180,E1 29132.195,E2 29132.195} C_VEL
LIN {X 0,Y 244.292,Z 1135.729,A -85,B 0,C 180,E1 29138.499,E2 29138.499} C_VEL
LIN {X 0,Y 271.02,Z 1102.499,A -85,B 0,C 180,E1 29142.982,E2 29142.982} C_VEL
LIN {X 0,Y 288.989,Z 1074.974,A -85,B 0,C 180,E1 29145.573,E2 29145.573} C_VEL
LIN {X 0,Y 290.931,Z 1062.025,A -85,B 0,C 180,E1 29151.009,E2 29151.009} C_VEL
LIN {X 0,Y 291.995,Z 1053.157,A -85,B 0,C 180,E1 29157.022,E2 29157.022} C_VEL
LIN {X 0,Y 293.123,Z 1049.029,A -85,B 0,C 180,E1 29162.958,E2 29162.958} C_VEL
LIN {X 0,Y 292.663,Z 1055.129,A -85,B 0,C 180,E1 29170.347,E2 29170.347} C_VEL
LIN {X 0,Y 292.313,Z 1064.226,A -85,B 0,C 180,E1 29175.784,E2 29175.784} C_VEL
LIN {X 0,Y 291.628,Z 1072.724,A -85,B 0,C 180,E1 29179.369,E2 29179.369} C_VEL
LIN {X 0,Y 286.621,Z 1081.477,A -85,B 0,C 180,E1 29180.18,E2 29180.18} C_VEL
LIN {X 0,Y 261.553,Z 1116.504,A -85,B 0,C 180,E1 29183.596,E2 29183.596} C_VEL
LIN {X 0,Y 234.657,Z 1146.582,A -85,B 0,C 180,E1 29188.379,E2 29188.379} C_VEL
LIN {X 0,Y 207.858,Z 1171.266,A -85,B 0,C 180,E1 29194.903,E2 29194.903} C_VEL
LIN {X 0,Y 181.2,Z 1192.052,A -85,B 0,C 180,E1 29204.699,E2 29204.699} C_VEL
LIN {X 0,Y 160.876,Z 1206.349,A -85,B 0,C 180,E1 29217.554,E2 29217.554} C_VEL
LIN {X 0,Y 149.522,Z 1214.43,A -85,B 0,C 180,E1 29232.301,E2 29232.301} C_VEL
LIN {X 0,Y 146.339,Z 1217.097,A -85,B 0,C 180,E1 29244.057,E2 29244.057} C_VEL
LIN {X 0,Y 146.172,Z 1217.292,A -85,B 0,C 180,E1 29252.042,E2 29252.042} C_VEL
LIN {X 0,Y 143.877,Z 1216.967,A -85,B 0,C 180,E1 29257.132,E2 29257.132} C_VEL
LIN {X 0,Y 140.49,Z 1215.595,A -85,B 0,C 180,E1 29264.988,E2 29264.988} C_VEL
LIN {X 0,Y 140.74,Z 1215.337,A -85,B 0,C 180,E1 29265.872,E2 29265.872} C_VEL
LIN {X 0,Y 151.734,Z 1208.033,A -85,B 0,C 180,E1 29281.736,E2 29281.736} C_VEL
LIN {X 0,Y 171.368,Z 1195.068,A -85,B 0,C 180,E1 29295.024,E2 29295.024} C_VEL
LIN {X 0,Y 196.305,Z 1176.925,A -85,B 0,C 180,E1 29304.77,E2 29304.77} C_VEL
LIN {X 0,Y 223.561,Z 1153.67,A -85,B 0,C 180,E1 29311.781,E2 29311.781} C_VEL
LIN {X 0,Y 251.501,Z 1124.745,A -85,B 0,C 180,E1 29316.878,E2 29316.878} C_VEL
LIN {X 0,Y 277.128,Z 1091.703,A -85,B 0,C 180,E1 29320.434,E2 29320.434} C_VEL
LIN {X 0,Y 286.491,Z 1077.409,A -85,B 0,C 180,E1 29321.507,E2 29321.507} C_VEL
LIN {X 0,Y 287.792,Z 1068.24,A -85,B 0,C 180,E1 29325.525,E2 29325.525} C_VEL
LIN {X 0,Y 288.228,Z 1060.234,A -85,B 0,C 180,E1 29330.932,E2 29330.932} C_VEL
LIN {X 0,Y 288.972,Z 1055.714,A -85,B 0,C 180,E1 29336.999,E2 29336.999} C_VEL
LIN {X 0,Y 287.993,Z 1058.178,A -85,B 0,C 180,E1 29341.392,E2 29341.392} C_VEL
LIN {X 0,Y 286.772,Z 1065.361,A -85,B 0,C 180,E1 29347.095,E2 29347.095} C_VEL
LIN {X 0,Y 284.749,Z 1076.297,A -85,B 0,C 180,E1 29352.291,E2 29352.291} C_VEL
LIN {X 0,Y 284.293,Z 1078.768,A -85,B 0,C 180,E1 29353.256,E2 29353.256} C_VEL
LIN {X 0,Y 257.898,Z 1115.91,A -85,B 0,C 180,E1 29356.923,E2 29356.923} C_VEL
LIN {X 0,Y 228.95,Z 1148.25,A -85,B 0,C 180,E1 29362.091,E2 29362.091} C_VEL
LIN {X 0,Y 199.86,Z 1175.047,A -85,B 0,C 180,E1 29369.328,E2 29369.328} C_VEL
LIN {X 0,Y 174.798,Z 1195.024,A -85,B 0,C 180,E1 29378.721,E2 29378.721} C_VEL
LIN {X 0,Y 153.608,Z 1210.652,A -85,B 0,C 180,E1 29392.101,E2 29392.101} C_VEL
LIN {X 0,Y 141.535,Z 1220.183,A -85,B 0,C 180,E1 29407.992,E2 29407.992} C_VEL
LIN {X 0,Y 137.973,Z 1224.303,A -85,B 0,C 180,E1 29423.694,E2 29423.694} C_VEL
LIN {X 0,Y 138.309,Z 1224.683,A -85,B 0,C 180,E1 29429.999,E2 29429.999} C_VEL
LIN {X 0,Y 138.645,Z 1223.236,A -85,B 0,C 180,E1 29442.625,E2 29442.625} C_VEL
LIN {X 0,Y 145.64,Z 1216.748,A -85,B 0,C 180,E1 29459.208,E2 29459.208} C_VEL
LIN {X 0,Y 160.444,Z 1205.699,A -85,B 0,C 180,E1 29473.212,E2 29473.212} C_VEL
LIN {X 0,Y 184.263,Z 1187.882,A -85,B 0,C 180,E1 29485.32,E2 29485.32} C_VEL
LIN {X 0,Y 212.586,Z 1164.129,A -85,B 0,C 180,E1 29494.143,E2 29494.143} C_VEL
LIN {X 0,Y 241.425,Z 1135.432,A -85,B 0,C 180,E1 29500.298,E2 29500.298} C_VEL
LIN {X 0,Y 268.594,Z 1102.349,A -85,B 0,C 180,E1 29504.618,E2 29504.618} C_VEL
LIN {X 0,Y 284.492,Z 1078.968,A -85,B 0,C 180,E1 29506.742,E2 29506.742} C_VEL
LIN {X 0,Y 286.844,Z 1066.477,A -85,B 0,C 180,E1 29512.407,E2 29512.407} C_VEL
LIN {X 0,Y 288.048,Z 1058.912,A -85,B 0,C 180,E1 29518.186,E2 29518.186} C_VEL
LIN {X 0,Y 289.183,Z 1055.996,A -85,B 0,C 180,E1 29522.999,E2 29522.999} C_VEL
LIN {X 0,Y 288.396,Z 1062.183,A -85,B 0,C 180,E1 29530.502,E2 29530.502} C_VEL
LIN {X 0,Y 287.615,Z 1071.782,A -85,B 0,C 180,E1 29536.05,E2 29536.05} C_VEL
LIN {X 0,Y 286.573,Z 1077.732,A -85,B 0,C 180,E1 29538.385,E2 29538.385} C_VEL
LIN {X 0,Y 262.488,Z 1111.837,A -85,B 0,C 180,E1 29541.431,E2 29541.431} C_VEL
LIN {X 0,Y 237.066,Z 1140.635,A -85,B 0,C 180,E1 29545.466,E2 29545.466} C_VEL
LIN {X 0,Y 210.365,Z 1165.614,A -85,B 0,C 180,E1 29551.2,E2 29551.2} C_VEL
LIN {X 0,Y 185.088,Z 1185.571,A -85,B 0,C 180,E1 29558.946,E2 29558.946} C_VEL
LIN {X 0,Y 161.335,Z 1201.959,A -85,B 0,C 180,E1 29570.657,E2 29570.657} C_VEL
LIN {X 0,Y 145.474,Z 1212.256,A -85,B 0,C 180,E1 29585.378,E2 29585.378} C_VEL
LIN {X 0,Y 139.564,Z 1216.345,A -85,B 0,C 180,E1 29597.621,E2 29597.621} C_VEL
LIN {X 0,Y 138.27,Z 1217.503,A -85,B 0,C 180,E1 29611.991,E2 29611.991} C_VEL
LIN {X 0,Y 140.74,Z 1215.337,A -85,B 0,C 180,E1 29625.872,E2 29625.872} C_VEL
LIN {X 0,Y 141.091,Z 1214.37,A -85,B 0,C 180,E1 29629.402,E2 29629.402} C_VEL
LIN {X 0,Y 140.981,Z 1210.737,A -85,B 0,C 180,E1 29639.171,E2 29639.171} C_VEL
LIN {X 0,Y 141.62,Z 1210.287,A -85,B 0,C 180,E1 29640.007,E2 29640.007} C_VEL
LIN {X 0,Y 160.931,Z 1198.426,A -85,B 0,C 180,E1 29654.482,E2 29654.482} C_VEL
LIN {X 0,Y 185.544,Z 1181.763,A -85,B 0,C 180,E1 29664.755,E2 29664.755} C_VEL
LIN {X 0,Y 212.522,Z 1160.387,A -85,B 0,C 180,E1 29672.065,E2 29672.065} C_VEL
LIN {X 0,Y 240.241,Z 1133.999,A -85,B 0,C 180,E1 29677.289,E2 29677.289} C_VEL
LIN {X 0,Y 267.248,Z 1102.108,A -85,B 0,C 180,E1 29681.118,E2 29681.118} C_VEL
LIN {X 0,Y 282.186,Z 1080.902,A -85,B 0,C 180,E1 29682.81,E2 29682.81} C_VEL
LIN {X 0,Y 283.534,Z 1071.336,A -85,B 0,C 180,E1 29687.664,E2 29687.664} C_VEL
LIN {X 0,Y 284.281,Z 1064.361,A -85,B 0,C 180,E1 29693.886,E2 29693.886} C_VEL
LIN {X 0,Y 284.801,Z 1062.492,A -85,B 0,C 180,E1 29696.955,E2 29696.955} C_VEL
LIN {X 0,Y 283.761,Z 1065.048,A -85,B 0,C 180,E1 29701.412,E2 29701.412} C_VEL
LIN {X 0,Y 282.205,Z 1071.992,A -85,B 0,C 180,E1 29706.941,E2 29706.941} C_VEL
LIN {X 0,Y 279.911,Z 1082.053,A -85,B 0,C 180,E1 29711.774,E2 29711.774} C_VEL
LIN {X 0,Y 275.549,Z 1088.973,A -85,B 0,C 180,E1 29712.556,E2 29712.556} C_VEL
LIN {X 0,Y 250.238,Z 1121.954,A -85,B 0,C 180,E1 29715.992,E2 29715.992} C_VEL
LIN {X 0,Y 222.859,Z 1150.955,A -85,B 0,C 180,E1 29720.785,E2 29720.785} C_VEL
LIN {X 0,Y 194.553,Z 1175.929,A -85,B 0,C 180,E1 29727.649,E2 29727.649} C_VEL
LIN {X 0,Y 167.451,Z 1196.457,A -85,B 0,C 180,E1 29737.645,E2 29737.645} C_VEL
LIN {X 0,Y 145.792,Z 1211.492,A -85,B 0,C 180,E1 29751.419,E2 29751.419} C_VEL
LIN {X 0,Y 134.096,Z 1219.975,A -85,B 0,C 180,E1 29766.702,E2 29766.702} C_VEL
LIN {X 0,Y 130.072,Z 1224.1,A -85,B 0,C 180,E1 29783.309,E2 29783.309} C_VEL
LIN {X 0,Y 130.388,Z 1224.48,A -85,B 0,C 180,E1 29789.999,E2 29789.999} C_VEL
LIN {X 0,Y 130.843,Z 1223.033,A -85,B 0,C 180,E1 29803.392,E2 29803.392} C_VEL
LIN {X 0,Y 137.768,Z 1217.161,A -85,B 0,C 180,E1 29819.674,E2 29819.674} C_VEL
LIN {X 0,Y 154.39,Z 1205.63,A -85,B 0,C 180,E1 29835.149,E2 29835.149} C_VEL
LIN {X 0,Y 179.704,Z 1187.651,A -85,B 0,C 180,E1 29847.48,E2 29847.48} C_VEL
LIN {X 0,Y 208.614,Z 1164.351,A -85,B 0,C 180,E1 29856.039,E2 29856.039} C_VEL
LIN {X 0,Y 237.808,Z 1136.229,A -85,B 0,C 180,E1 29861.97,E2 29861.97} C_VEL
LIN {X 0,Y 265.334,Z 1103.677,A -85,B 0,C 180,E1 29866.13,E2 29866.13} C_VEL
LIN {X 0,Y 279.013,Z 1084.282,A -85,B 0,C 180,E1 29867.838,E2 29867.838} C_VEL
LIN {X 0,Y 280.303,Z 1081.586,A -85,B 0,C 180,E1 29868.485,E2 29868.485} C_VEL
LIN {X 0,Y 282.658,Z 1070.989,A -85,B 0,C 180,E1 29873.842,E2 29873.842} C_VEL
LIN {X 0,Y 284.305,Z 1064.199,A -85,B 0,C 180,E1 29879.996,E2 29879.996} C_VEL
LIN {X 0,Y 284.997,Z 1062.801,A -85,B 0,C 180,E1 29883.043,E2 29883.043} C_VEL
LIN {X 0,Y 284.216,Z 1067.493,A -85,B 0,C 180,E1 29889.197,E2 29889.197} C_VEL
LIN {X 0,Y 283.112,Z 1076.208,A -85,B 0,C 180,E1 29894.859,E2 29894.859} C_VEL
LIN {X 0,Y 282.446,Z 1080.755,A -85,B 0,C 180,E1 29896.953,E2 29896.953} C_VEL
LIN {X 0,Y 256.441,Z 1116.184,A -85,B 0,C 180,E1 29900.241,E2 29900.241} C_VEL
LIN {X 0,Y 229.075,Z 1145.634,A -85,B 0,C 180,E1 29904.559,E2 29904.559} C_VEL
LIN {X 0,Y 199.134,Z 1171.716,A -85,B 0,C 180,E1 29911.124,E2 29911.124} C_VEL
LIN {X 0,Y 170.295,Z 1192.475,A -85,B 0,C 180,E1 29920.859,E2 29920.859} C_VEL
LIN {X 0,Y 149.672,Z 1205.522,A -85,B 0,C 180,E1 29932.596,E2 29932.596} C_VEL
LIN {X 0,Y 134.432,Z 1214.839,A -85,B 0,C 180,E1 29950.236,E2 29950.236} C_VEL
LIN {X 0,Y 130.605,Z 1217.501,A -85,B 0,C 180,E1 29963.338,E2 29963.338} C_VEL
LIN {X 0,Y 130.53,Z 1217.812,A -85,B 0,C 180,E1 29970.001,E2 29970.001} C_VEL
LIN {X 0,Y 132.949,Z 1215.641,A -85,B 0,C 180,E1 29986.431,E2 29986.431} C_VEL
LIN {X 0,Y 141.62,Z 1210.287,A -85,B 0,C 180,E1 30000.007,E2 30000.007} C_VEL
LIN {X 0,Y 144.567,Z 1206.68,A -85,B 0,C 180,E1 30006.778,E2 30006.778} C_VEL
LIN {X 0,Y 149.277,Z 1202.279,A -85,B 0,C 180,E1 30013.157,E2 30013.157} C_VEL
LIN {X 0,Y 175.604,Z 1185.788,A -85,B 0,C 180,E1 30025.062,E2 30025.062} C_VEL
LIN {X 0,Y 206.081,Z 1163.069,A -85,B 0,C 180,E1 30033.381,E2 30033.381} C_VEL
LIN {X 0,Y 235.658,Z 1136.018,A -85,B 0,C 180,E1 30038.806,E2 30038.806} C_VEL
LIN {X 0,Y 263.949,Z 1103.613,A -85,B 0,C 180,E1 30042.635,E2 30042.635} C_VEL
LIN {X 0,Y 277.636,Z 1084.589,A -85,B 0,C 180,E1 30044.172,E2 30044.172} C_VEL
LIN {X 0,Y 279.297,Z 1075.075,A -85,B 0,C 180,E1 30049.772,E2 30049.772} C_VEL
LIN {X 0,Y 279.905,Z 1071.15,A -85,B 0,C 180,E1 30053.79,E2 30053.79} C_VEL
LIN {X 0,Y 280.532,Z 1069.262,A -85,B 0,C 180,E1 30056.909,E2 30056.909} C_VEL
LIN {X 0,Y 279.283,Z 1071.919,A -85,B 0,C 180,E1 30061.558,E2 30061.558} C_VEL
LIN {X 0,Y 277.435,Z 1079.063,A -85,B 0,C 180,E1 30067.062,E2 30067.062} C_VEL
LIN {X 0,Y 275.394,Z 1086.176,A -85,B 0,C 180,E1 30070.599,E2 30070.599} C_VEL
LIN {X 0,Y 251.504,Z 1117.729,A -85,B 0,C 180,E1 30073.706,E2 30073.706} C_VEL
LIN {X 0,Y 223.333,Z 1147.717,A -85,B 0,C 180,E1 30078.214,E2 30078.214} C_VEL
LIN {X 0,Y 192.396,Z 1174.566,A -85,B 0,C 180,E1 30085.077,E2 30085.077} C_VEL
LIN {X 0,Y 162.576,Z 1196.236,A -85,B 0,C 180,E1 30095.358,E2 30095.358} C_VEL
LIN {X 0,Y 139.053,Z 1211.544,A -85,B 0,C 180,E1 30109.707,E2 30109.707} C_VEL
LIN {X 0,Y 125.206,Z 1221.01,A -85,B 0,C 180,E1 30128.71,E2 30128.71} C_VEL
LIN {X 0,Y 122.178,Z 1223.896,A -85,B 0,C 180,E1 30142.875,E2 30142.875} C_VEL
LIN {X 0,Y 122.467,Z 1224.278,A -85,B 0,C 180,E1 30149.999,E2 30149.999} C_VEL
LIN {X 0,Y 123.081,Z 1222.829,A -85,B 0,C 180,E1 30164.253,E2 30164.253} C_VEL
LIN {X 0,Y 130.777,Z 1216.956,A -85,B 0,C 180,E1 30181.426,E2 30181.426} C_VEL
LIN {X 0,Y 148.596,Z 1205.51,A -85,B 0,C 180,E1 30197.289,E2 30197.289} C_VEL
LIN {X 0,Y 175.432,Z 1187.422,A -85,B 0,C 180,E1 30209.739,E2 30209.739} C_VEL
LIN {X 0,Y 205.263,Z 1164.248,A -85,B 0,C 180,E1 30218.081,E2 30218.081} C_VEL
LIN {X 0,Y 234.682,Z 1136.721,A -85,B 0,C 180,E1 30223.736,E2 30223.736} C_VEL
LIN {X 0,Y 263.506,Z 1103.31,A -85,B 0,C 180,E1 30227.844,E2 30227.844} C_VEL
LIN {X 0,Y 275.355,Z 1086.917,A -85,B 0,C 180,E1 30229.236,E2 30229.236} C_VEL
LIN {X 0,Y 277.961,Z 1077.939,A -85,B 0,C 180,E1 30233.738,E2 30233.738} C_VEL
LIN {X 0,Y 279.942,Z 1070.929,A -85,B 0,C 180,E1 30239.996,E2 30239.996} C_VEL
LIN {X 0,Y 280.728,Z 1069.546,A -85,B 0,C 180,E1 30243.089,E2 30243.089} C_VEL
LIN {X 0,Y 279.476,Z 1075.416,A -85,B 0,C 180,E1 30250.221,E2 30250.221} C_VEL
LIN {X 0,Y 277.881,Z 1084.449,A -85,B 0,C 180,E1 30255.562,E2 30255.562} C_VEL
LIN {X 0,Y 262.155,Z 1106.248,A -85,B 0,C 180,E1 30257.5,E2 30257.5} C_VEL
LIN {X 0,Y 233.921,Z 1138.001,A -85,B 0,C 180,E1 30261.381,E2 30261.381} C_VEL
LIN {X 0,Y 204.074,Z 1164.892,A -85,B 0,C 180,E1 30266.999,E2 30266.999} C_VEL
LIN {X 0,Y 175.479,Z 1185.999,A -85,B 0,C 180,E1 30274.882,E2 30274.882} C_VEL
LIN {X 0,Y 149.312,Z 1202.371,A -85,B 0,C 180,E1 30286.764,E2 30286.764} C_VEL
LIN {X 0,Y 131.13,Z 1212.667,A -85,B 0,C 180,E1 30302.47,E2 30302.47} C_VEL
LIN {X 0,Y 123.141,Z 1217.271,A -85,B 0,C 180,E1 30319.735,E2 30319.735} C_VEL
LIN {X 0,Y 122.622,Z 1218.014,A -85,B 0,C 180,E1 30330.001,E2 30330.001} C_VEL
LIN {X 0,Y 124.201,Z 1216.665,A -85,B 0,C 180,E1 30344.124,E2 30344.124} C_VEL
LIN {X 0,Y 134.286,Z 1210.763,A -85,B 0,C 180,E1 30361.193,E2 30361.193} C_VEL
LIN {X 0,Y 149.277,Z 1202.279,A -85,B 0,C 180,E1 30373.157,E2 30373.157} C_VEL
LIN {X 0,Y 155.42,Z 1197.201,A -85,B 0,C 180,E1 30379.039,E2 30379.039} C_VEL
LIN {X 0,Y 162.827,Z 1191.239,A -85,B 0,C 180,E1 30384.352,E2 30384.352} C_VEL
LIN {X 0,Y 192.954,Z 1170.772,A -85,B 0,C 180,E1 30393.291,E2 30393.291} C_VEL
LIN {X 0,Y 224.646,Z 1144.22,A -85,B 0,C 180,E1 30399.376,E2 30399.376} C_VEL
LIN {X 0,Y 253.982,Z 1113.37,A -85,B 0,C 180,E1 30403.399,E2 30403.399} C_VEL
LIN {X 0,Y 272.453,Z 1089.548,A -85,B 0,C 180,E1 30405.403,E2 30405.403} C_VEL
LIN {X 0,Y 273.792,Z 1085.491,A -85,B 0,C 180,E1 30407.218,E2 30407.218} C_VEL
LIN {X 0,Y 275.162,Z 1078.906,A -85,B 0,C 180,E1 30412.416,E2 30412.416} C_VEL
LIN {X 0,Y 276.032,Z 1075.885,A -85,B 0,C 180,E1 30416.858,E2 30416.858} C_VEL
LIN {X 0,Y 274.737,Z 1078.604,A -85,B 0,C 180,E1 30421.584,E2 30421.584} C_VEL
LIN {X 0,Y 272.789,Z 1084.609,A -85,B 0,C 180,E1 30426.381,E2 30426.381} C_VEL
LIN {X 0,Y 271.046,Z 1090.069,A -85,B 0,C 180,E1 30429.252,E2 30429.252} C_VEL
LIN {X 0,Y 244.127,Z 1123.72,A -85,B 0,C 180,E1 30432.636,E2 30432.636} C_VEL
LIN {X 0,Y 214.327,Z 1153.394,A -85,B 0,C 180,E1 30437.358,E2 30437.358} C_VEL
LIN {X 0,Y 184.533,Z 1177.659,A -85,B 0,C 180,E1 30444.001,E2 30444.001} C_VEL
LIN {X 0,Y 155.443,Z 1197.594,A -85,B 0,C 180,E1 30454.043,E2 30454.043} C_VEL
LIN {X 0,Y 133.401,Z 1211.067,A -85,B 0,C 180,E1 30467.035,E2 30467.035} C_VEL
LIN {X 0,Y 117.723,Z 1220.803,A -85,B 0,C 180,E1 30487.284,E2 30487.284} C_VEL
LIN {X 0,Y 114.328,Z 1223.694,A -85,B 0,C 180,E1 30502.383,E2 30502.383} C_VEL
LIN {X 0,Y 114.571,Z 1224.076,A -85,B 0,C 180,E1 30509.999,E2 30509.999} C_VEL
LIN {X 0,Y 115.328,Z 1222.625,A -85,B 0,C 180,E1 30525.234,E2 30525.234} C_VEL
LIN {X 0,Y 123.907,Z 1216.746,A -85,B 0,C 180,E1 30543.388,E2 30543.388} C_VEL
LIN {X 0,Y 144.044,Z 1204.75,A -85,B 0,C 180,E1 30560.21,E2 30560.21} C_VEL
LIN {X 0,Y 171.461,Z 1187.193,A -85,B 0,C 180,E1 30572.097,E2 30572.097} C_VEL
LIN {X 0,Y 201.65,Z 1164.603,A -85,B 0,C 180,E1 30580.07,E2 30580.07} C_VEL
LIN {X 0,Y 232.877,Z 1136.077,A -85,B 0,C 180,E1 30585.703,E2 30585.703} C_VEL
LIN {X 0,Y 261.921,Z 1102.942,A -85,B 0,C 180,E1 30589.576,E2 30589.576} C_VEL
LIN {X 0,Y 271.261,Z 1090.234,A -85,B 0,C 180,E1 30590.755,E2 30590.755} C_VEL
LIN {X 0,Y 273.723,Z 1082.512,A -85,B 0,C 180,E1 30595.17,E2 30595.17} C_VEL
LIN {X 0,Y 275.441,Z 1077.546,A -85,B 0,C 180,E1 30599.996,E2 30599.996} C_VEL
LIN {X 0,Y 276.231,Z 1076.164,A -85,B 0,C 180,E1 30603.139,E2 30603.139} C_VEL
LIN {X 0,Y 274.98,Z 1081.205,A -85,B 0,C 180,E1 30609.509,E2 30609.509} C_VEL
LIN {X 0,Y 273.421,Z 1088.109,A -85,B 0,C 180,E1 30614.042,E2 30614.042} C_VEL
LIN {X 0,Y 271.116,Z 1091.936,A -85,B 0,C 180,E1 30614.649,E2 30614.649} C_VEL
LIN {X 0,Y 242.86,Z 1126.317,A -85,B 0,C 180,E1 30617.919,E2 30617.919} C_VEL
LIN {X 0,Y 213.215,Z 1154.798,A -85,B 0,C 180,E1 30622.499,E2 30622.499} C_VEL
LIN {X 0,Y 182.452,Z 1178.582,A -85,B 0,C 180,E1 30629.304,E2 30629.304} C_VEL
LIN {X 0,Y 151.933,Z 1197.862,A -85,B 0,C 180,E1 30640.173,E2 30640.173} C_VEL
LIN {X 0,Y 129.15,Z 1210.24,A -85,B 0,C 180,E1 30655.177,E2 30655.177} C_VEL
LIN {X 0,Y 116.446,Z 1216.92,A -85,B 0,C 180,E1 30674.916,E2 30674.916} C_VEL
LIN {X 0,Y 114.733,Z 1218.216,A -85,B 0,C 180,E1 30690.001,E2 30690.001} C_VEL
LIN {X 0,Y 116.509,Z 1216.869,A -85,B 0,C 180,E1 30705.078,E2 30705.078} C_VEL
LIN {X 0,Y 129.538,Z 1209.989,A -85,B 0,C 180,E1 30725.069,E2 30725.069} C_VEL
LIN {X 0,Y 152.417,Z 1197.479,A -85,B 0,C 180,E1 30739.979,E2 30739.979} C_VEL
LIN {X 0,Y 162.827,Z 1191.239,A -85,B 0,C 180,E1 30744.352,E2 30744.352} C_VEL
LIN {X 0,Y 171.384,Z 1184.716,A -85,B 0,C 180,E1 30749.106,E2 30749.106} C_VEL
LIN {X 0,Y 180.562,Z 1177.285,A -85,B 0,C 180,E1 30753.337,E2 30753.337} C_VEL
LIN {X 0,Y 212.023,Z 1153.274,A -85,B 0,C 180,E1 30759.724,E2 30759.724} C_VEL
LIN {X 0,Y 242.332,Z 1124.308,A -85,B 0,C 180,E1 30764.029,E2 30764.029} C_VEL
LIN {X 0,Y 268.662,Z 1092.499,A -85,B 0,C 180,E1 30766.97,E2 30766.97} C_VEL
LIN {X 0,Y 270.372,Z 1085.437,A -85,B 0,C 180,E1 30772.368,E2 30772.368} C_VEL
LIN {X 0,Y 271.431,Z 1082.436,A -85,B 0,C 180,E1 30776.805,E2 30776.805} C_VEL
LIN {X 0,Y 269.94,Z 1085.156,A -85,B 0,C 180,E1 30781.612,E2 30781.612} C_VEL
LIN {X 0,Y 267.677,Z 1091.49,A -85,B 0,C 180,E1 30786.504,E2 30786.504} C_VEL
LIN {X 0,Y 266.744,Z 1093.906,A -85,B 0,C 180,E1 30787.836,E2 30787.836} C_VEL
LIN {X 0,Y 238.957,Z 1127.266,A -85,B 0,C 180,E1 30791.229,E2 30791.229} C_VEL
LIN {X 0,Y 207.05,Z 1157.47,A -85,B 0,C 180,E1 30796.145,E2 30796.145} C_VEL
LIN {X 0,Y 174.803,Z 1182.114,A -85,B 0,C 180,E1 30803.398,E2 30803.398} C_VEL
LIN {X 0,Y 143.877,Z 1201.635,A -85,B 0,C 180,E1 30814.668,E2 30814.668} C_VEL
LIN {X 0,Y 120.279,Z 1214.839,A -85,B 0,C 180,E1 30830.955,E2 30830.955} C_VEL
LIN {X 0,Y 110.328,Z 1220.597,A -85,B 0,C 180,E1 30845.666,E2 30845.666} C_VEL
LIN {X 0,Y 106.298,Z 1223.7,A -85,B 0,C 180,E1 30866.187,E2 30866.187} C_VEL
LIN {X 0,Y 106.298,Z 1223.707,A -85,B 0,C 180,E1 30873.811,E2 30873.811} C_VEL
LIN {X 0,Y 110.343,Z 1220.633,A -85,B 0,C 180,E1 30894.328,E2 30894.328} C_VEL
LIN {X 0,Y 127.546,Z 1210.937,A -85,B 0,C 180,E1 30915.464,E2 30915.464} C_VEL
LIN {X 0,Y 153.689,Z 1195.927,A -85,B 0,C 180,E1 30929.62,E2 30929.62} C_VEL
LIN {X 0,Y 186.035,Z 1174.276,A -85,B 0,C 180,E1 30939.503,E2 30939.503} C_VEL
LIN {X 0,Y 218.786,Z 1147.445,A -85,B 0,C 180,E1 30945.84,E2 30945.84} C_VEL
LIN {X 0,Y 249.941,Z 1115.486,A -85,B 0,C 180,E1 30950.119,E2 30950.119} C_VEL
LIN {X 0,Y 266.091,Z 1095.355,A -85,B 0,C 180,E1 30951.919,E2 30951.919} C_VEL
LIN {X 0,Y 267.894,Z 1091.668,A -85,B 0,C 180,E1 30953.502,E2 30953.502} C_VEL
LIN {X 0,Y 270.106,Z 1085.431,A -85,B 0,C 180,E1 30958.389,E2 30958.389} C_VEL
LIN {X 0,Y 271.624,Z 1082.699,A -85,B 0,C 180,E1 30963.193,E2 30963.193} C_VEL
LIN {X 0,Y 270.044,Z 1087.884,A -85,B 0,C 180,E1 30969.684,E2 30969.684} C_VEL
LIN {X 0,Y 268.208,Z 1093.669,A -85,B 0,C 180,E1 30973.12,E2 30973.12} C_VEL
LIN {X 0,Y 240.534,Z 1126.6,A -85,B 0,C 180,E1 30976.117,E2 30976.117} C_VEL
LIN {X 0,Y 209.015,Z 1156.075,A -85,B 0,C 180,E1 30980.708,E2 30980.708} C_VEL
LIN {X 0,Y 178.675,Z 1178.809,A -85,B 0,C 180,E1 30987.068,E2 30987.068} C_VEL
LIN {X 0,Y 148.479,Z 1197.216,A -85,B 0,C 180,E1 30997.079,E2 30997.079} C_VEL
LIN {X 0,Y 123.592,Z 1209.987,A -85,B 0,C 180,E1 31012.193,E2 31012.193} C_VEL
LIN {X 0,Y 112.251,Z 1215.45,A -85,B 0,C 180,E1 31026.111,E2 31026.111} C_VEL
LIN {X 0,Y 107.013,Z 1218.126,A -85,B 0,C 180,E1 31042.196,E2 31042.196} C_VEL
LIN {X 0,Y 106.824,Z 1218.418,A -85,B 0,C 180,E1 31050.001,E2 31050.001} C_VEL
LIN {X 0,Y 108.858,Z 1217.073,A -85,B 0,C 180,E1 31066.166,E2 31066.166} C_VEL
LIN {X 0,Y 119.699,Z 1211.759,A -85,B 0,C 180,E1 31083.864,E2 31083.864} C_VEL
LIN {X 0,Y 142.459,Z 1200.289,A -85,B 0,C 180,E1 31100.047,E2 31100.047} C_VEL
LIN {X 0,Y 171.253,Z 1183.446,A -85,B 0,C 180,E1 31110.837,E2 31110.837} C_VEL
LIN {X 0,Y 180.562,Z 1177.285,A -85,B 0,C 180,E1 31113.337,E2 31113.337} C_VEL
LIN {X 0,Y 190.401,Z 1169.247,A -85,B 0,C 180,E1 31117.086,E2 31117.086} C_VEL
LIN {X 0,Y 199.172,Z 1161.75,A -85,B 0,C 180,E1 31120.065,E2 31120.065} C_VEL
LIN {X 0,Y 200.693,Z 1160.518,A -85,B 0,C 180,E1 31120.353,E2 31120.353} C_VEL
LIN {X 0,Y 230.037,Z 1134.98,A -85,B 0,C 180,E1 31124.635,E2 31124.635} C_VEL
LIN {X 0,Y 259.625,Z 1102.427,A -85,B 0,C 180,E1 31127.854,E2 31127.854} C_VEL
LIN {X 0,Y 263.184,Z 1097.857,A -85,B 0,C 180,E1 31128.178,E2 31128.178} C_VEL
LIN {X 0,Y 264.414,Z 1095.491,A -85,B 0,C 180,E1 31129.172,E2 31129.172} C_VEL
LIN {X 0,Y 266.149,Z 1089.841,A -85,B 0,C 180,E1 31135.107,E2 31135.107} C_VEL
LIN {X 0,Y 266.634,Z 1088.854,A -85,B 0,C 180,E1 31136.747,E2 31136.747} C_VEL
LIN {X 0,Y 265.065,Z 1091.672,A -85,B 0,C 180,E1 31141.642,E2 31141.642} C_VEL
LIN {X 0,Y 262.835,Z 1096.819,A -85,B 0,C 180,E1 31145.793,E2 31145.793} C_VEL
LIN {X 0,Y 261.922,Z 1098.617,A -85,B 0,C 180,E1 31146.647,E2 31146.647} C_VEL
LIN {X 0,Y 234.045,Z 1130.46,A -85,B 0,C 180,E1 31149.74,E2 31149.74} C_VEL
LIN {X 0,Y 203.237,Z 1158.568,A -85,B 0,C 180,E1 31154.243,E2 31154.243} C_VEL
LIN {X 0,Y 171.013,Z 1182.33,A -85,B 0,C 180,E1 31161.069,E2 31161.069} C_VEL
LIN {X 0,Y 139.443,Z 1201.386,A -85,B 0,C 180,E1 31171.869,E2 31171.869} C_VEL
LIN {X 0,Y 114.098,Z 1214.63,A -85,B 0,C 180,E1 31188.391,E2 31188.391} C_VEL
LIN {X 0,Y 103.027,Z 1220.391,A -85,B 0,C 180,E1 31203.816,E2 31203.816} C_VEL
LIN {X 0,Y 98.562,Z 1223.287,A -85,B 0,C 180,E1 31221.155,E2 31221.155} C_VEL
LIN {X 0,Y 98.731,Z 1223.671,A -85,B 0,C 180,E1 31229.999,E2 31229.999} C_VEL
LIN {X 0,Y 99.935,Z 1222.216,A -85,B 0,C 180,E1 31247.652,E2 31247.652} C_VEL
LIN {X 0,Y 110.694,Z 1216.33,A -85,B 0,C 180,E1 31268.024,E2 31268.024} C_VEL
LIN {X 0,Y 131.143,Z 1205.99,A -85,B 0,C 180,E1 31283.979,E2 31283.979} C_VEL
LIN {X 0,Y 161.409,Z 1188.688,A -85,B 0,C 180,E1 31296.25,E2 31296.25} C_VEL
LIN {X 0,Y 195.542,Z 1165.021,A -85,B 0,C 180,E1 31304.329,E2 31304.329} C_VEL
LIN {X 0,Y 229.154,Z 1135.737,A -85,B 0,C 180,E1 31309.612,E2 31309.612} C_VEL
LIN {X 0,Y 259.471,Z 1102.205,A -85,B 0,C 180,E1 31313.111,E2 31313.111} C_VEL
LIN {X 0,Y 261.946,Z 1099.014,A -85,B 0,C 180,E1 31313.354,E2 31313.354} C_VEL
LIN {X 0,Y 264.042,Z 1094.633,A -85,B 0,C 180,E1 31315.883,E2 31315.883} C_VEL
LIN {X 0,Y 265.925,Z 1090.497,A -85,B 0,C 180,E1 31319.996,E2 31319.996} C_VEL
LIN {X 0,Y 266.816,Z 1089.129,A -85,B 0,C 180,E1 31323.25,E2 31323.25} C_VEL
LIN {X 0,Y 264.95,Z 1094.578,A -85,B 0,C 180,E1 31329.872,E2 31329.872} C_VEL
LIN {X 0,Y 264.337,Z 1096.455,A -85,B 0,C 180,E1 31331.255,E2 31331.255} C_VEL
LIN {X 0,Y 262.236,Z 1099.518,A -85,B 0,C 180,E1 31331.847,E2 31331.847} C_VEL
LIN {X 0,Y 234.969,Z 1130.352,A -85,B 0,C 180,E1 31334.686,E2 31334.686} C_VEL
LIN {X 0,Y 205.388,Z 1157.053,A -85,B 0,C 180,E1 31338.786,E2 31338.786} C_VEL
LIN {X 0,Y 175.185,Z 1179.034,A -85,B 0,C 180,E1 31344.741,E2 31344.741} C_VEL
LIN {X 0,Y 142.375,Z 1198.151,A -85,B 0,C 180,E1 31355.116,E2 31355.116} C_VEL
LIN {X 0,Y 117.366,Z 1210.194,A -85,B 0,C 180,E1 31369.795,E2 31369.795} C_VEL
LIN {X 0,Y 105.008,Z 1215.655,A -85,B 0,C 180,E1 31384.349,E2 31384.349} C_VEL
LIN {X 0,Y 99.189,Z 1218.31,A -85,B 0,C 180,E1 31401.214,E2 31401.214} C_VEL
LIN {X 0,Y 98.936,Z 1218.62,A -85,B 0,C 180,E1 31410.001,E2 31410.001} C_VEL
LIN {X 0,Y 101.246,Z 1217.277,A -85,B 0,C 180,E1 31427.418,E2 31427.418} C_VEL
LIN {X 0,Y 114.459,Z 1211.387,A -85,B 0,C 180,E1 31447.445,E2 31447.445} C_VEL
LIN {X 0,Y 139.604,Z 1199.419,A -85,B 0,C 180,E1 31463.58,E2 31463.58} C_VEL
LIN {X 0,Y 169.095,Z 1182.666,A -85,B 0,C 180,E1 31473.654,E2 31473.654} C_VEL
LIN {X 0,Y 200.693,Z 1160.518,A -85,B 0,C 180,E1 31480.353,E2 31480.353} C_VEL
LIN {X 0,Y 211.224,Z 1151.106,A -85,B 0,C 180,E1 31483.246,E2 31483.246} C_VEL
LIN {X 0,Y 221.777,Z 1141.055,A -85,B 0,C 180,E1 31485.823,E2 31485.823} C_VEL
LIN {X 0,Y 250.407,Z 1111.839,A -85,B 0,C 180,E1 31488.883,E2 31488.883} C_VEL
LIN {X 0,Y 259.491,Z 1100.823,A -85,B 0,C 180,E1 31489.918,E2 31489.918} C_VEL
LIN {X 0,Y 261.085,Z 1096.342,A -85,B 0,C 180,E1 31494.704,E2 31494.704} C_VEL
LIN {X 0,Y 261.698,Z 1095.187,A -85,B 0,C 180,E1 31496.686,E2 31496.686} C_VEL
LIN {X 0,Y 259.913,Z 1098.011,A -85,B 0,C 180,E1 31501.675,E2 31501.675} C_VEL
LIN {X 0,Y 258.114,Z 1101.872,A -85,B 0,C 180,E1 31504.886,E2 31504.886} C_VEL
LIN {X 0,Y 253.989,Z 1107.037,A -85,B 0,C 180,E1 31505.544,E2 31505.544} C_VEL
LIN {X 0,Y 224.266,Z 1138.518,A -85,B 0,C 180,E1 31508.821,E2 31508.821} C_VEL
LIN {X 0,Y 192.643,Z 1165.175,A -85,B 0,C 180,E1 31513.46,E2 31513.46} C_VEL
LIN {X 0,Y 158.286,Z 1188.316,A -85,B 0,C 180,E1 31521.03,E2 31521.03} C_VEL
LIN {X 0,Y 126.527,Z 1205.664,A -85,B 0,C 180,E1 31533.035,E2 31533.035} C_VEL
LIN {X 0,Y 101.106,Z 1217.664,A -85,B 0,C 180,E1 31553.165,E2 31553.165} C_VEL
LIN {X 0,Y 92.314,Z 1221.987,A -85,B 0,C 180,E1 31570.834,E2 31570.834} C_VEL
LIN {X 0,Y 90.823,Z 1223.469,A -85,B 0,C 180,E1 31589.999,E2 31589.999} C_VEL
LIN {X 0,Y 92.315,Z 1222.012,A -85,B 0,C 180,E1 31609.164,E2 31609.164} C_VEL
LIN {X 0,Y 104.403,Z 1216.121,A -85,B 0,C 180,E1 31630.776,E2 31630.776} C_VEL
LIN {X 0,Y 126.513,Z 1205.776,A -85,B 0,C 180,E1 31646.971,E2 31646.971} C_VEL
LIN {X 0,Y 158.298,Z 1188.468,A -85,B 0,C 180,E1 31658.955,E2 31658.955} C_VEL
LIN {X 0,Y 192.564,Z 1165.469,A -85,B 0,C 180,E1 31666.491,E2 31666.491} C_VEL
LIN {X 0,Y 226.039,Z 1137.186,A -85,B 0,C 180,E1 31671.411,E2 31671.411} C_VEL
LIN {X 0,Y 256.837,Z 1104.099,A -85,B 0,C 180,E1 31674.73,E2 31674.73} C_VEL
LIN {X 0,Y 258.192,Z 1102.323,A -85,B 0,C 180,E1 31674.948,E2 31674.948} C_VEL
LIN {X 0,Y 260.884,Z 1096.801,A -85,B 0,C 180,E1 31679.995,E2 31679.995} C_VEL
LIN {X 0,Y 261.882,Z 1095.435,A -85,B 0,C 180,E1 31683.312,E2 31683.312} C_VEL
LIN {X 0,Y 260.008,Z 1100.044,A -85,B 0,C 180,E1 31689.181,E2 31689.181} C_VEL
LIN {X 0,Y 259.619,Z 1101.159,A -85,B 0,C 180,E1 31690.077,E2 31690.077} C_VEL
LIN {X 0,Y 231.924,Z 1131.777,A -85,B 0,C 180,E1 31692.926,E2 31692.926} C_VEL
LIN {X 0,Y 201.506,Z 1158.417,A -85,B 0,C 180,E1 31696.885,E2 31696.885} C_VEL
LIN {X 0,Y 168.777,Z 1181.184,A -85,B 0,C 180,E1 31703.039,E2 31703.039} C_VEL
LIN {X 0,Y 138.647,Z 1198.023,A -85,B 0,C 180,E1 31712.117,E2 31712.117} C_VEL
LIN {X 0,Y 111.368,Z 1210.4,A -85,B 0,C 180,E1 31727.133,E2 31727.133} C_VEL
LIN {X 0,Y 97.878,Z 1215.859,A -85,B 0,C 180,E1 31742.327,E2 31742.327} C_VEL
LIN {X 0,Y 90.911,Z 1218.78,A -85,B 0,C 180,E1 31768.338,E2 31768.338} C_VEL
LIN {X 0,Y 93.701,Z 1217.481,A -85,B 0,C 180,E1 31788.872,E2 31788.872} C_VEL
LIN {X 0,Y 108.211,Z 1211.594,A -85,B 0,C 180,E1 31810.024,E2 31810.024} C_VEL
LIN {X 0,Y 133.423,Z 1200.396,A -85,B 0,C 180,E1 31825.63,E2 31825.63} C_VEL
LIN {X 0,Y 163.002,Z 1184.547,A -85,B 0,C 180,E1 31835.445,E2 31835.445} C_VEL
LIN {X 0,Y 195.195,Z 1163.063,A -85,B 0,C 180,E1 31842.045,E2 31842.045} C_VEL
LIN {X 0,Y 221.777,Z 1141.055,A -85,B 0,C 180,E1 31845.823,E2 31845.823} C_VEL
LIN {X 0,Y 232.342,Z 1130.34,A -85,B 0,C 180,E1 31848.108,E2 31848.108} C_VEL
LIN {X 0,Y 241.333,Z 1120.56,A -85,B 0,C 180,E1 31849.972,E2 31849.972} C_VEL
LIN {X 0,Y 242.775,Z 1119.016,A -85,B 0,C 180,E1 31850.122,E2 31850.122} C_VEL
LIN {X 0,Y 254.846,Z 1105.324,A -85,B 0,C 180,E1 31851.365,E2 31851.365} C_VEL
LIN {X 0,Y 256.601,Z 1101.4,A -85,B 0,C 180,E1 31856.62,E2 31856.62} C_VEL
LIN {X 0,Y 254.707,Z 1104.324,A -85,B 0,C 180,E1 31861.709,E2 31861.709} C_VEL
LIN {X 0,Y 253.663,Z 1106.188,A -85,B 0,C 180,E1 31863.428,E2 31863.428} C_VEL
LIN {X 0,Y 248.018,Z 1112.826,A -85,B 0,C 180,E1 31864.193,E2 31864.193} C_VEL
LIN {X 0,Y 217.734,Z 1143.117,A -85,B 0,C 180,E1 31867.379,E2 31867.379} C_VEL
LIN {X 0,Y 185.836,Z 1168.502,A -85,B 0,C 180,E1 31871.908,E2 31871.908} C_VEL
LIN {X 0,Y 152.308,Z 1189.874,A -85,B 0,C 180,E1 31879.064,E2 31879.064} C_VEL
LIN {X 0,Y 119.534,Z 1206.662,A -85,B 0,C 180,E1 31891.164,E2 31891.164} C_VEL
LIN {X 0,Y 94.723,Z 1217.455,A -85,B 0,C 180,E1 31910.215,E2 31910.215} C_VEL
LIN {X 0,Y 84.767,Z 1221.781,A -85,B 0,C 180,E1 31929.051,E2 31929.051} C_VEL
LIN {X 0,Y 82.892,Z 1223.266,A -85,B 0,C 180,E1 31949.999,E2 31949.999} C_VEL
LIN {X 0,Y 84.768,Z 1221.807,A -85,B 0,C 180,E1 31970.946,E2 31970.946} C_VEL
LIN {X 0,Y 98.394,Z 1215.911,A -85,B 0,C 180,E1 31993.868,E2 31993.868} C_VEL
LIN {X 0,Y 124.756,Z 1204.328,A -85,B 0,C 180,E1 32011.343,E2 32011.343} C_VEL
LIN {X 0,Y 155.55,Z 1188.248,A -85,B 0,C 180,E1 32021.766,E2 32021.766} C_VEL
LIN {X 0,Y 191.053,Z 1165.06,A -85,B 0,C 180,E1 32028.921,E2 32028.921} C_VEL
LIN {X 0,Y 224.97,Z 1136.91,A -85,B 0,C 180,E1 32033.455,E2 32033.455} C_VEL
LIN {X 0,Y 252.473,Z 1108.091,A -85,B 0,C 180,E1 32036.199,E2 32036.199} C_VEL
LIN {X 0,Y 253.824,Z 1106.41,A -85,B 0,C 180,E1 32036.574,E2 32036.574} C_VEL
LIN {X 0,Y 255.751,Z 1103.047,A -85,B 0,C 180,E1 32039.995,E2 32039.995} C_VEL
LIN {X 0,Y 256.794,Z 1101.635,A -85,B 0,C 180,E1 32043.377,E2 32043.377} C_VEL
LIN {X 0,Y 255.043,Z 1105.46,A -85,B 0,C 180,E1 32048.466,E2 32048.466} C_VEL
LIN {X 0,Y 253.091,Z 1107.866,A -85,B 0,C 180,E1 32048.918,E2 32048.918} C_VEL
LIN {X 0,Y 223.311,Z 1138.639,A -85,B 0,C 180,E1 32051.737,E2 32051.737} C_VEL
LIN {X 0,Y 190.421,Z 1165.304,A -85,B 0,C 180,E1 32056.026,E2 32056.026} C_VEL
LIN {X 0,Y 157.671,Z 1186.217,A -85,B 0,C 180,E1 32062.355,E2 32062.355} C_VEL
LIN {X 0,Y 123.186,Z 1203.415,A -85,B 0,C 180,E1 32073.914,E2 32073.914} C_VEL
LIN {X 0,Y 97.461,Z 1213.696,A -85,B 0,C 180,E1 32091.546,E2 32091.546} C_VEL
LIN {X 0,Y 86.159,Z 1217.731,A -85,B 0,C 180,E1 32109.407,E2 32109.407} C_VEL
LIN {X 0,Y 83.155,Z 1219.023,A -85,B 0,C 180,E1 32130.001,E2 32130.001} C_VEL
LIN {X 0,Y 86.213,Z 1217.685,A -85,B 0,C 180,E1 32150.582,E2 32150.582} C_VEL
LIN {X 0,Y 102.106,Z 1211.841,A -85,B 0,C 180,E1 32172.818,E2 32172.818} C_VEL
LIN {X 0,Y 127.484,Z 1201.346,A -85,B 0,C 180,E1 32187.903,E2 32187.903} C_VEL
LIN {X 0,Y 160.691,Z 1184.273,A -85,B 0,C 180,E1 32198.245,E2 32198.245} C_VEL
LIN {X 0,Y 194.553,Z 1162.047,A -85,B 0,C 180,E1 32204.547,E2 32204.547} C_VEL
LIN {X 0,Y 227.182,Z 1134.752,A -85,B 0,C 180,E1 32208.603,E2 32208.603} C_VEL
LIN {X 0,Y 242.775,Z 1119.016,A -85,B 0,C 180,E1 32210.122,E2 32210.122} C_VEL
LIN {X 0,Y 247.394,Z 1113.586,A -85,B 0,C 180,E1 32211.34,E2 32211.34} C_VEL
LIN {X 0,Y 250.341,Z 1109.164,A -85,B 0,C 180,E1 32213.98,E2 32213.98} C_VEL
LIN {X 0,Y 250.707,Z 1108.539,A -85,B 0,C 180,E1 32214.699,E2 32214.699} C_VEL
LIN {X 0,Y 251.345,Z 1107.488,A -85,B 0,C 180,E1 32216.549,E2 32216.549} C_VEL
LIN {X 0,Y 249.245,Z 1110.381,A -85,B 0,C 180,E1 32221.665,E2 32221.665} C_VEL
LIN {X 0,Y 247.974,Z 1112.009,A -85,B 0,C 180,E1 32222.292,E2 32222.292} C_VEL
LIN {X 0,Y 218.675,Z 1141.213,A -85,B 0,C 180,E1 32225.052,E2 32225.052} C_VEL
LIN {X 0,Y 186.101,Z 1167.035,A -85,B 0,C 180,E1 32229.154,E2 32229.154} C_VEL
LIN {X 0,Y 153.187,Z 1187.863,A -85,B 0,C 180,E1 32235.321,E2 32235.321} C_VEL
LIN {X 0,Y 118.404,Z 1205.227,A -85,B 0,C 180,E1 32246.382,E2 32246.382} C_VEL
LIN {X 0,Y 88.628,Z 1217.246,A -85,B 0,C 180,E1 32266.85,E2 32266.85} C_VEL
LIN {X 0,Y 77.33,Z 1221.576,A -85,B 0,C 180,E1 32286.926,E2 32286.926} C_VEL
LIN {X 0,Y 74.97,Z 1223.064,A -85,B 0,C 180,E1 32309.998,E2 32309.998} C_VEL
LIN {X 0,Y 77.33,Z 1221.603,A -85,B 0,C 180,E1 32333.071,E2 32333.071} C_VEL
LIN {X 0,Y 92.699,Z 1215.703,A -85,B 0,C 180,E1 32357.355,E2 32357.355} C_VEL
LIN {X 0,Y 121.333,Z 1203.973,A -85,B 0,C 180,E1 32374.88,E2 32374.88} C_VEL
LIN {X 0,Y 156.55,Z 1186.051,A -85,B 0,C 180,E1 32385.447,E2 32385.447} C_VEL
LIN {X 0,Y 191.46,Z 1163.462,A -85,B 0,C 180,E1 32391.607,E2 32391.607} C_VEL
LIN {X 0,Y 226.028,Z 1134.857,A -85,B 0,C 180,E1 32395.719,E2 32395.719} C_VEL
LIN {X 0,Y 248.043,Z 1112.336,A -85,B 0,C 180,E1 32397.71,E2 32397.71} C_VEL
LIN {X 0,Y 249.622,Z 1110.27,A -85,B 0,C 180,E1 32398.662,E2 32398.662} C_VEL
LIN {X 0,Y 251.525,Z 1107.715,A -85,B 0,C 180,E1 32403.448,E2 32403.448} C_VEL
LIN {X 0,Y 250.218,Z 1110.071,A -85,B 0,C 180,E1 32406.95,E2 32406.95} C_VEL
LIN {X 0,Y 247.646,Z 1113.139,A -85,B 0,C 180,E1 32407.469,E2 32407.469} C_VEL
LIN {X 0,Y 215.639,Z 1144.362,A -85,B 0,C 180,E1 32410.338,E2 32410.338} C_VEL
LIN {X 0,Y 180.872,Z 1170.655,A -85,B 0,C 180,E1 32414.795,E2 32414.795} C_VEL
LIN {X 0,Y 146.627,Z 1190.707,A -85,B 0,C 180,E1 32421.553,E2 32421.553} C_VEL
LIN {X 0,Y 114.94,Z 1205.187,A -85,B 0,C 180,E1 32432.499,E2 32432.499} C_VEL
LIN {X 0,Y 91.341,Z 1213.901,A -85,B 0,C 180,E1 32448.428,E2 32448.428} C_VEL
LIN {X 0,Y 78.766,Z 1217.934,A -85,B 0,C 180,E1 32467.373,E2 32467.373} C_VEL
LIN {X 0,Y 75.263,Z 1219.225,A -85,B 0,C 180,E1 32490.001,E2 32490.001} C_VEL
LIN {X 0,Y 78.817,Z 1217.889,A -85,B 0,C 180,E1 32512.615,E2 32512.615} C_VEL
LIN {X 0,Y 96.862,Z 1211.887,A -85,B 0,C 180,E1 32536.441,E2 32536.441} C_VEL
LIN {X 0,Y 127.85,Z 1199.601,A -85,B 0,C 180,E1 32552.739,E2 32552.739} C_VEL
LIN {X 0,Y 159.911,Z 1183.342,A -85,B 0,C 180,E1 32561.369,E2 32561.369} C_VEL
LIN {X 0,Y 194.346,Z 1160.984,A -85,B 0,C 180,E1 32567.064,E2 32567.064} C_VEL
LIN {X 0,Y 226.656,Z 1134.172,A -85,B 0,C 180,E1 32570.661,E2 32570.661} C_VEL
LIN {X 0,Y 248.945,Z 1111.252,A -85,B 0,C 180,E1 32572.553,E2 32572.553} C_VEL
LIN {X 0,Y 250.106,Z 1109.758,A -85,B 0,C 180,E1 32573.047,E2 32573.047} C_VEL
LIN {X 0,Y 250.707,Z 1108.539,A -85,B 0,C 180,E1 32574.699,E2 32574.699} C_VEL
LIN {X 0,Y 249.249,Z 1109.809,A -85,B 0,C 180,E1 32576.616,E2 32576.616} C_VEL
LIN {X 0,Y 244.85,Z 1114.802,A -85,B 0,C 180,E1 32579.802,E2 32579.802} C_VEL
LIN {X 0,Y 243.521,Z 1116.378,A -85,B 0,C 180,E1 32580.741,E2 32580.741} C_VEL
LIN {X 0,Y 210.315,Z 1147.638,A -85,B 0,C 180,E1 32583.688,E2 32583.688} C_VEL
LIN {X 0,Y 175.157,Z 1173.406,A -85,B 0,C 180,E1 32588.054,E2 32588.054} C_VEL
LIN {X 0,Y 138.513,Z 1194.263,A -85,B 0,C 180,E1 32595.259,E2 32595.259} C_VEL
LIN {X 0,Y 103.11,Z 1209.787,A -85,B 0,C 180,E1 32608.143,E2 32608.143} C_VEL
LIN {X 0,Y 75.389,Z 1219.563,A -85,B 0,C 180,E1 32632.914,E2 32632.914} C_VEL
LIN {X 0,Y 67.22,Z 1222.471,A -85,B 0,C 180,E1 32656.971,E2 32656.971} C_VEL
LIN {X 0,Y 67.035,Z 1222.861,A -85,B 0,C 180,E1 32669.998,E2 32669.998} C_VEL
LIN {X 0,Y 70,Z 1221.398,A -85,B 0,C 180,E1 32695.653,E2 32695.653} C_VEL
LIN {X 0,Y 87.365,Z 1215.507,A -85,B 0,C 180,E1 32721.249,E2 32721.249} C_VEL
LIN {X 0,Y 118.099,Z 1203.757,A -85,B 0,C 180,E1 32738.467,E2 32738.467} C_VEL
LIN {X 0,Y 151.231,Z 1187.803,A -85,B 0,C 180,E1 32747.664,E2 32747.664} C_VEL
LIN {X 0,Y 188.62,Z 1164.554,A -85,B 0,C 180,E1 32753.798,E2 32753.798} C_VEL
LIN {X 0,Y 223.699,Z 1136.339,A -85,B 0,C 180,E1 32757.608,E2 32757.608} C_VEL
LIN {X 0,Y 243.587,Z 1116.687,A -85,B 0,C 180,E1 32759.259,E2 32759.259} C_VEL
LIN {X 0,Y 244.948,Z 1115.138,A -85,B 0,C 180,E1 32759.995,E2 32759.995} C_VEL
LIN {X 0,Y 246.142,Z 1113.701,A -85,B 0,C 180,E1 32763.524,E2 32763.524} C_VEL
LIN {X 0,Y 245.35,Z 1114.993,A -85,B 0,C 180,E1 32765.584,E2 32765.584} C_VEL
LIN {X 0,Y 212.536,Z 1146.209,A -85,B 0,C 180,E1 32768.421,E2 32768.421} C_VEL
LIN {X 0,Y 176.211,Z 1172.708,A -85,B 0,C 180,E1 32772.724,E2 32772.724} C_VEL
LIN {X 0,Y 140.541,Z 1192.638,A -85,B 0,C 180,E1 32779.37,E2 32779.37} C_VEL
LIN {X 0,Y 106.199,Z 1207.189,A -85,B 0,C 180,E1 32791.12,E2 32791.12} C_VEL
LIN {X 0,Y 77.49,Z 1216.471,A -85,B 0,C 180,E1 32814.083,E2 32814.083} C_VEL
LIN {X 0,Y 68.013,Z 1219.12,A -85,B 0,C 180,E1 32837.129,E2 32837.129} C_VEL
LIN {X 0,Y 67.349,Z 1219.427,A -85,B 0,C 180,E1 32850.002,E2 32850.002} C_VEL
LIN {X 0,Y 71.539,Z 1218.094,A -85,B 0,C 180,E1 32875.065,E2 32875.065} C_VEL
LIN {X 0,Y 90.233,Z 1212.497,A -85,B 0,C 180,E1 32899.088,E2 32899.088} C_VEL
LIN {X 0,Y 121.255,Z 1201.129,A -85,B 0,C 180,E1 32914.963,E2 32914.963} C_VEL
LIN {X 0,Y 154.512,Z 1185.268,A -85,B 0,C 180,E1 32923.531,E2 32923.531} C_VEL
LIN {X 0,Y 190.926,Z 1162.545,A -85,B 0,C 180,E1 32929.16,E2 32929.16} C_VEL
LIN {X 0,Y 224.314,Z 1135.592,A -85,B 0,C 180,E1 32932.55,E2 32932.55} C_VEL
LIN {X 0,Y 243.887,Z 1116.185,A -85,B 0,C 180,E1 32934.117,E2 32934.117} C_VEL
LIN {X 0,Y 245.26,Z 1114.624,A -85,B 0,C 180,E1 32934.539,E2 32934.539} C_VEL
LIN {X 0,Y 245.965,Z 1113.471,A -85,B 0,C 180,E1 32936.474,E2 32936.474} C_VEL
LIN {X 0,Y 244.85,Z 1114.802,A -85,B 0,C 180,E1 32939.802,E2 32939.802} C_VEL
LIN {X 0,Y 242.419,Z 1117.436,A -85,B 0,C 180,E1 32940.45,E2 32940.45} C_VEL
LIN {X 0,Y 228.013,Z 1131.472,A -85,B 0,C 180,E1 32939.928,E2 32939.928} C_VEL
LIN {X 0,Y 195.342,Z 1158.656,A -85,B 0,C 180,E1 32942.873,E2 32942.873} C_VEL
LIN {X 0,Y 160.438,Z 1181.436,A -85,B 0,C 180,E1 32947.382,E2 32947.382} C_VEL
LIN {X 0,Y 121.979,Z 1200.667,A -85,B 0,C 180,E1 32955.685,E2 32955.685} C_VEL
LIN {X 0,Y 87.906,Z 1213.577,A -85,B 0,C 180,E1 32970.469,E2 32970.469} C_VEL
LIN {X 0,Y 69.094,Z 1219.356,A -85,B 0,C 180,E1 32988.856,E2 32988.856} C_VEL
LIN {X 0,Y 59.476,Z 1222.267,A -85,B 0,C 180,E1 33015.238,E2 33015.238} C_VEL
LIN {X 0,Y 59.114,Z 1222.659,A -85,B 0,C 180,E1 33029.998,E2 33029.998} C_VEL
LIN {X 0,Y 62.859,Z 1221.193,A -85,B 0,C 180,E1 33058.822,E2 33058.822} C_VEL
LIN {X 0,Y 85.345,Z 1214.418,A -85,B 0,C 180,E1 33087.809,E2 33087.809} C_VEL
LIN {X 0,Y 118.641,Z 1202.167,A -85,B 0,C 180,E1 33103.313,E2 33103.313} C_VEL
LIN {X 0,Y 153.254,Z 1185.6,A -85,B 0,C 180,E1 33111.391,E2 33111.391} C_VEL
LIN {X 0,Y 189.76,Z 1162.956,A -85,B 0,C 180,E1 33116.519,E2 33116.519} C_VEL
LIN {X 0,Y 224.75,Z 1134.881,A -85,B 0,C 180,E1 33119.787,E2 33119.787} C_VEL
LIN {X 0,Y 238.407,Z 1121.7,A -85,B 0,C 180,E1 33120.801,E2 33120.801} C_VEL
LIN {X 0,Y 239.711,Z 1120.343,A -85,B 0,C 180,E1 33121.197,E2 33121.197} C_VEL
LIN {X 0,Y 240.377,Z 1119.763,A -85,B 0,C 180,E1 33124.06,E2 33124.06} C_VEL
LIN {X 0,Y 207.837,Z 1149.366,A -85,B 0,C 180,E1 33126.608,E2 33126.608} C_VEL
LIN {X 0,Y 173.488,Z 1173.611,A -85,B 0,C 180,E1 33130.311,E2 33130.311} C_VEL
LIN {X 0,Y 138.097,Z 1192.852,A -85,B 0,C 180,E1 33136.241,E2 33136.241} C_VEL
LIN {X 0,Y 102.286,Z 1207.399,A -85,B 0,C 180,E1 33147.273,E2 33147.273} C_VEL
LIN {X 0,Y 71.182,Z 1216.675,A -85,B 0,C 180,E1 33170.312,E2 33170.312} C_VEL
LIN {X 0,Y 60.314,Z 1219.322,A -85,B 0,C 180,E1 33195.451,E2 33195.451} C_VEL
LIN {X 0,Y 59.434,Z 1219.629,A -85,B 0,C 180,E1 33210.002,E2 33210.002} C_VEL
LIN {X 0,Y 64.42,Z 1218.298,A -85,B 0,C 180,E1 33238.065,E2 33238.065} C_VEL
LIN {X 0,Y 85.209,Z 1212.702,A -85,B 0,C 180,E1 33263.156,E2 33263.156} C_VEL
LIN {X 0,Y 118.086,Z 1201.339,A -85,B 0,C 180,E1 33278.488,E2 33278.488} C_VEL
LIN {X 0,Y 152.036,Z 1185.712,A -85,B 0,C 180,E1 33286.351,E2 33286.351} C_VEL
LIN {X 0,Y 189.588,Z 1162.791,A -85,B 0,C 180,E1 33291.528,E2 33291.528} C_VEL
LIN {X 0,Y 224.142,Z 1135.208,A -85,B 0,C 180,E1 33294.621,E2 33294.621} C_VEL
LIN {X 0,Y 240.24,Z 1119.513,A -85,B 0,C 180,E1 33295.937,E2 33295.937} C_VEL
LIN {X 0,Y 239.61,Z 1120.058,A -85,B 0,C 180,E1 33298.71,E2 33298.71} C_VEL
LIN {X 0,Y 236.916,Z 1122.841,A -85,B 0,C 180,E1 33299.276,E2 33299.276} C_VEL
LIN {X 0,Y 228.013,Z 1131.472,A -85,B 0,C 180,E1 33299.928,E2 33299.928} C_VEL
LIN {X 0,Y 214.784,Z 1143.114,A -85,B 0,C 180,E1 33299.916,E2 33299.916} C_VEL
LIN {X 0,Y 201.087,Z 1153.981,A -85,B 0,C 180,E1 33299.958,E2 33299.958} C_VEL
LIN {X 0,Y 163.289,Z 1179.086,A -85,B 0,C 180,E1 33303.975,E2 33303.975} C_VEL
LIN {X 0,Y 123.515,Z 1198.977,A -85,B 0,C 180,E1 33311.049,E2 33311.049} C_VEL
LIN {X 0,Y 84.058,Z 1213.365,A -85,B 0,C 180,E1 33325.662,E2 33325.662} C_VEL
LIN {X 0,Y 59.357,Z 1220.029,A -85,B 0,C 180,E1 33349.995,E2 33349.995} C_VEL
LIN {X 0,Y 51.78,Z 1222.062,A -85,B 0,C 180,E1 33372.982,E2 33372.982} C_VEL
LIN {X 0,Y 51.173,Z 1222.456,A -85,B 0,C 180,E1 33389.998,E2 33389.998} C_VEL
LIN {X 0,Y 55.935,Z 1220.988,A -85,B 0,C 180,E1 33422.804,E2 33422.804} C_VEL
LIN {X 0,Y 80.505,Z 1214.428,A -85,B 0,C 180,E1 33452.179,E2 33452.179} C_VEL
LIN {X 0,Y 116.556,Z 1201.955,A -85,B 0,C 180,E1 33467.167,E2 33467.167} C_VEL
LIN {X 0,Y 152.245,Z 1185.374,A -85,B 0,C 180,E1 33474.434,E2 33474.434} C_VEL
LIN {X 0,Y 189.439,Z 1162.704,A -85,B 0,C 180,E1 33478.995,E2 33478.995} C_VEL
LIN {X 0,Y 224.867,Z 1134.588,A -85,B 0,C 180,E1 33481.86,E2 33481.86} C_VEL
LIN {X 0,Y 234,Z 1126.098,A -85,B 0,C 180,E1 33482.457,E2 33482.457} C_VEL
LIN {X 0,Y 199.492,Z 1155.524,A -85,B 0,C 180,E1 33485.041,E2 33485.041} C_VEL
LIN {X 0,Y 161.115,Z 1180.355,A -85,B 0,C 180,E1 33489.062,E2 33489.062} C_VEL
LIN {X 0,Y 122.155,Z 1199.06,A -85,B 0,C 180,E1 33495.982,E2 33495.982} C_VEL
LIN {X 0,Y 86.448,Z 1211.436,A -85,B 0,C 180,E1 33508.789,E2 33508.789} C_VEL
LIN {X 0,Y 57.463,Z 1218.544,A -85,B 0,C 180,E1 33538.172,E2 33538.172} C_VEL
LIN {X 0,Y 51.519,Z 1219.831,A -85,B 0,C 180,E1 33570.002,E2 33570.002} C_VEL
LIN {X 0,Y 57.519,Z 1218.502,A -85,B 0,C 180,E1 33601.797,E2 33601.797} C_VEL
LIN {X 0,Y 80.673,Z 1212.906,A -85,B 0,C 180,E1 33627.701,E2 33627.701} C_VEL
LIN {X 0,Y 115.387,Z 1201.549,A -85,B 0,C 180,E1 33642.196,E2 33642.196} C_VEL
LIN {X 0,Y 150.352,Z 1185.936,A -85,B 0,C 180,E1 33649.31,E2 33649.31} C_VEL
LIN {X 0,Y 188.578,Z 1163.04,A -85,B 0,C 180,E1 33653.926,E2 33653.926} C_VEL
LIN {X 0,Y 223.883,Z 1135.178,A -85,B 0,C 180,E1 33656.664,E2 33656.664} C_VEL
LIN {X 0,Y 234.163,Z 1125.554,A -85,B 0,C 180,E1 33657.499,E2 33657.499} C_VEL
LIN {X 0,Y 201.087,Z 1153.981,A -85,B 0,C 180,E1 33659.958,E2 33659.958} C_VEL
LIN {X 0,Y 186.858,Z 1164.234,A -85,B 0,C 180,E1 33660.029,E2 33660.029} C_VEL
LIN {X 0,Y 172.02,Z 1173.529,A -85,B 0,C 180,E1 33660.158,E2 33660.158} C_VEL
LIN {X 0,Y 133.199,Z 1194.025,A -85,B 0,C 180,E1 33665.239,E2 33665.239} C_VEL
LIN {X 0,Y 94.064,Z 1209.142,A -85,B 0,C 180,E1 33674.856,E2 33674.856} C_VEL
LIN {X 0,Y 57.876,Z 1218.94,A -85,B 0,C 180,E1 33698.235,E2 33698.235} C_VEL
LIN {X 0,Y 44.188,Z 1221.858,A -85,B 0,C 180,E1 33729.942,E2 33729.942} C_VEL
LIN {X 0,Y 43.247,Z 1222.253,A -85,B 0,C 180,E1 33749.997,E2 33749.997} C_VEL
LIN {X 0,Y 49.377,Z 1220.783,A -85,B 0,C 180,E1 33787.86,E2 33787.86} C_VEL
LIN {X 0,Y 74.24,Z 1214.958,A -85,B 0,C 180,E1 33815.896,E2 33815.896} C_VEL
LIN {X 0,Y 111.452,Z 1203.116,A -85,B 0,C 180,E1 33830.293,E2 33830.293} C_VEL
LIN {X 0,Y 149.253,Z 1186.43,A -85,B 0,C 180,E1 33837.187,E2 33837.187} C_VEL
LIN {X 0,Y 187.564,Z 1163.797,A -85,B 0,C 180,E1 33841.301,E2 33841.301} C_VEL
LIN {X 0,Y 202.097,Z 1153.359,A -85,B 0,C 180,E1 33842.402,E2 33842.402} C_VEL
LIN {X 0,Y 165.59,Z 1177.416,A -85,B 0,C 180,E1 33845.648,E2 33845.648} C_VEL
LIN {X 0,Y 129.164,Z 1195.528,A -85,B 0,C 180,E1 33850.579,E2 33850.579} C_VEL
LIN {X 0,Y 96.008,Z 1207.817,A -85,B 0,C 180,E1 33858.746,E2 33858.746} C_VEL
LIN {X 0,Y 59.784,Z 1217.082,A -85,B 0,C 180,E1 33880.505,E2 33880.505} C_VEL
LIN {X 0,Y 45.123,Z 1219.728,A -85,B 0,C 180,E1 33910.381,E2 33910.381} C_VEL
LIN {X 0,Y 43.607,Z 1220.034,A -85,B 0,C 180,E1 33930.003,E2 33930.003} C_VEL
LIN {X 0,Y 50.933,Z 1218.706,A -85,B 0,C 180,E1 33966.516,E2 33966.516} C_VEL
LIN {X 0,Y 82.947,Z 1211.538,A -85,B 0,C 180,E1 33995.984,E2 33995.984} C_VEL
LIN {X 0,Y 120.241,Z 1199.122,A -85,B 0,C 180,E1 34007.602,E2 34007.602} C_VEL
LIN {X 0,Y 161.916,Z 1179.343,A -85,B 0,C 180,E1 34013.91,E2 34013.91} C_VEL
LIN {X 0,Y 199.598,Z 1154.996,A -85,B 0,C 180,E1 34017.221,E2 34017.221} C_VEL
LIN {X 0,Y 201.532,Z 1153.503,A -85,B 0,C 180,E1 34017.351,E2 34017.351} C_VEL
LIN {X 0,Y 185.662,Z 1164.838,A -85,B 0,C 180,E1 34018.855,E2 34018.855} C_VEL
LIN {X 0,Y 172.02,Z 1173.529,A -85,B 0,C 180,E1 34020.158,E2 34020.158} C_VEL
LIN {X 0,Y 156.702,Z 1182.134,A -85,B 0,C 180,E1 34020.345,E2 34020.345} C_VEL
LIN {X 0,Y 141.045,Z 1189.907,A -85,B 0,C 180,E1 34020.609,E2 34020.609} C_VEL
LIN {X 0,Y 100.326,Z 1206.285,A -85,B 0,C 180,E1 34027.762,E2 34027.762} C_VEL
LIN {X 0,Y 65.194,Z 1216.2,A -85,B 0,C 180,E1 34041.604,E2 34041.604} C_VEL
LIN {X 0,Y 43.291,Z 1220.547,A -85,B 0,C 180,E1 34065.566,E2 34065.566} C_VEL
LIN {X 0,Y 35.298,Z 1222.05,A -85,B 0,C 180,E1 34109.997,E2 34109.997} C_VEL
LIN {X 0,Y 45.003,Z 1220.244,A -85,B 0,C 180,E1 34157.647,E2 34157.647} C_VEL
LIN {X 0,Y 78.374,Z 1213.026,A -85,B 0,C 180,E1 34185.169,E2 34185.169} C_VEL
LIN {X 0,Y 117.732,Z 1200.154,A -85,B 0,C 180,E1 34195.914,E2 34195.914} C_VEL
LIN {X 0,Y 159.151,Z 1180.946,A -85,B 0,C 180,E1 34201.392,E2 34201.392} C_VEL
LIN {X 0,Y 166.789,Z 1176.624,A -85,B 0,C 180,E1 34202.074,E2 34202.074} C_VEL
LIN {X 0,Y 166.868,Z 1176.57,A -85,B 0,C 180,E1 34202.715,E2 34202.715} C_VEL
LIN {X 0,Y 130.874,Z 1194.531,A -85,B 0,C 180,E1 34206.638,E2 34206.638} C_VEL
LIN {X 0,Y 93.744,Z 1208.025,A -85,B 0,C 180,E1 34214.111,E2 34214.111} C_VEL
LIN {X 0,Y 54.931,Z 1217.286,A -85,B 0,C 180,E1 34234.155,E2 34234.155} C_VEL
LIN {X 0,Y 37.738,Z 1219.93,A -85,B 0,C 180,E1 34266.329,E2 34266.329} C_VEL
LIN {X 0,Y 35.69,Z 1220.236,A -85,B 0,C 180,E1 34290.003,E2 34290.003} C_VEL
LIN {X 0,Y 44.786,Z 1218.91,A -85,B 0,C 180,E1 34332.588,E2 34332.588} C_VEL
LIN {X 0,Y 80.021,Z 1211.746,A -85,B 0,C 180,E1 34361.233,E2 34361.233} C_VEL
LIN {X 0,Y 118.784,Z 1199.332,A -85,B 0,C 180,E1 34371.364,E2 34371.364} C_VEL
LIN {X 0,Y 161.265,Z 1179.575,A -85,B 0,C 180,E1 34376.724,E2 34376.724} C_VEL
LIN {X 0,Y 166.88,Z 1176.35,A -85,B 0,C 180,E1 34377.223,E2 34377.223} C_VEL
LIN {X 0,Y 166.796,Z 1176.407,A -85,B 0,C 180,E1 34377.898,E2 34377.898} C_VEL
LIN {X 0,Y 141.045,Z 1189.907,A -85,B 0,C 180,E1 34380.609,E2 34380.609} C_VEL
LIN {X 0,Y 124.95,Z 1196.894,A -85,B 0,C 180,E1 34380.983,E2 34380.983} C_VEL
LIN {X 0,Y 108.566,Z 1203.03,A -85,B 0,C 180,E1 34381.469,E2 34381.469} C_VEL
LIN {X 0,Y 70.357,Z 1214.2,A -85,B 0,C 180,E1 34391.223,E2 34391.223} C_VEL
LIN {X 0,Y 37.966,Z 1220.341,A -85,B 0,C 180,E1 34417.033,E2 34417.033} C_VEL
LIN {X 0,Y 27.353,Z 1221.847,A -85,B 0,C 180,E1 34469.996,E2 34469.996} C_VEL
LIN {X 0,Y 37.962,Z 1220.372,A -85,B 0,C 180,E1 34522.964,E2 34522.964} C_VEL
LIN {X 0,Y 76.693,Z 1212.816,A -85,B 0,C 180,E1 34551.068,E2 34551.068} C_VEL
LIN {X 0,Y 118.071,Z 1199.71,A -85,B 0,C 180,E1 34559.99,E2 34559.99} C_VEL
LIN {X 0,Y 136.5,Z 1192.015,A -85,B 0,C 180,E1 34562.463,E2 34562.463} C_VEL
LIN {X 0,Y 95.747,Z 1207.106,A -85,B 0,C 180,E1 34568.466,E2 34568.466} C_VEL
LIN {X 0,Y 57.272,Z 1216.321,A -85,B 0,C 180,E1 34582.182,E2 34582.182} C_VEL
LIN {X 0,Y 30.631,Z 1220.133,A -85,B 0,C 180,E1 34620.354,E2 34620.354} C_VEL
LIN {X 0,Y 27.784,Z 1220.438,A -85,B 0,C 180,E1 34650.004,E2 34650.004} C_VEL
LIN {X 0,Y 39.305,Z 1219.114,A -85,B 0,C 180,E1 34700.453,E2 34700.453} C_VEL
LIN {X 0,Y 77.815,Z 1211.955,A -85,B 0,C 180,E1 34726.825,E2 34726.825} C_VEL
LIN {X 0,Y 117.542,Z 1199.651,A -85,B 0,C 180,E1 34735.173,E2 34735.173} C_VEL
LIN {X 0,Y 136.481,Z 1191.857,A -85,B 0,C 180,E1 34737.774,E2 34737.774} C_VEL
LIN {X 0,Y 108.566,Z 1203.03,A -85,B 0,C 180,E1 34741.469,E2 34741.469} C_VEL
LIN {X 0,Y 102.005,Z 1205.237,A -85,B 0,C 180,E1 34740.8,E2 34740.8} C_VEL
LIN {X 0,Y 89.814,Z 1208.723,A -85,B 0,C 180,E1 34735.445,E2 34735.445} C_VEL
LIN {X 0,Y 88.386,Z 1209.089,A -85,B 0,C 180,E1 34735.123,E2 34735.123} C_VEL
LIN {X 0,Y 47.186,Z 1217.734,A -85,B 0,C 180,E1 34721.3,E2 34721.3} C_VEL
LIN {X 0,Y 24.088,Z 1220.317,A -85,B 0,C 180,E1 34688.986,E2 34688.986} C_VEL
LIN {X 0,Y 19.865,Z 1220.64,A -85,B 0,C 180,E1 34650.006,E2 34650.006} C_VEL
LIN {X 0,Y 46.386,Z 1217.876,A -85,B 0,C 180,E1 34579.034,E2 34579.034} C_VEL
LIN {X 0,Y 88.222,Z 1209.229,A -85,B 0,C 180,E1 34564.823,E2 34564.823} C_VEL
LIN {X 0,Y 102.39,Z 1205.064,A -85,B 0,C 180,E1 34562.029,E2 34562.029} C_VEL
LIN {X 0,Y 61.097,Z 1215.849,A -85,B 0,C 180,E1 34552.76,E2 34552.76} C_VEL
LIN {X 0,Y 32.251,Z 1220.305,A -85,B 0,C 180,E1 34531.942,E2 34531.942} C_VEL
LIN {X 0,Y 19.398,Z 1221.644,A -85,B 0,C 180,E1 34469.994,E2 34469.994} C_VEL
LIN {X 0,Y 33.731,Z 1220.134,A -85,B 0,C 180,E1 34406.035,E2 34406.035} C_VEL
LIN {X 0,Y 68.433,Z 1214.167,A -85,B 0,C 180,E1 34384.824,E2 34384.824} C_VEL
LIN {X 0,Y 102.543,Z 1204.901,A -85,B 0,C 180,E1 34377.946,E2 34377.946} C_VEL
LIN {X 0,Y 88.386,Z 1209.089,A -85,B 0,C 180,E1 34375.123,E2 34375.123} C_VEL
LIN {X 0,Y 71.435,Z 1213.24,A -85,B 0,C 180,E1 34374.72,E2 34374.72} C_VEL
LIN {X 0,Y 54.319,Z 1216.509,A -85,B 0,C 180,E1 34374.123,E2 34374.123} C_VEL
LIN {X 0,Y 18.6,Z 1220.52,A -85,B 0,C 180,E1 34344.567,E2 34344.567} C_VEL
LIN {X 0,Y 11.969,Z 1220.842,A -85,B 0,C 180,E1 34290.009,E2 34290.009} C_VEL
LIN {X 0,Y 31.619,Z 1219.559,A -85,B 0,C 180,E1 34216.585,E2 34216.585} C_VEL
LIN {X 0,Y 68.192,Z 1214.042,A -85,B 0,C 180,E1 34202.014,E2 34202.014} C_VEL
LIN {X 0,Y 31.039,Z 1219.961,A -85,B 0,C 180,E1 34187.505,E2 34187.505} C_VEL
LIN {X 0,Y 11.439,Z 1221.44,A -85,B 0,C 180,E1 34109.99,E2 34109.99} C_VEL
LIN {X 0,Y 31.044,Z 1219.927,A -85,B 0,C 180,E1 34032.499,E2 34032.499} C_VEL
LIN {X 0,Y 68.402,Z 1213.921,A -85,B 0,C 180,E1 34017.953,E2 34017.953} C_VEL
LIN {X 0,Y 54.319,Z 1216.509,A -85,B 0,C 180,E1 34014.123,E2 34014.123} C_VEL
LIN {X 0,Y 45.239,Z 1217.952,A -85,B 0,C 180,E1 34012.686,E2 34012.686} C_VEL
LIN {X 0,Y 19.665,Z 1220.446,A -85,B 0,C 180,E1 34012.839,E2 34012.839} C_VEL
LIN {X 0,Y 17.389,Z 1220.593,A -85,B 0,C 180,E1 34011.345,E2 34011.345} C_VEL
LIN {X 0,Y 4.047,Z 1221.045,A -85,B 0,C 180,E1 33930.028,E2 33930.028} C_VEL
LIN {X 0,Y 28.842,Z 1219.868,A -85,B 0,C 180,E1 33842.045,E2 33842.045} C_VEL
LIN {X 0,Y 3.476,Z 1221.237,A -85,B 0,C 180,E1 33749.968,E2 33749.968} C_VEL
LIN {X 0,Y 28.931,Z 1219.834,A -85,B 0,C 180,E1 33657.906,E2 33657.906} C_VEL
LIN {X 0,Y 17.389,Z 1220.593,A -85,B 0,C 180,E1 33651.345,E2 33651.345} C_VEL
LIN {X 0,Y 15.587,Z 1222.589,A -85,B 0,C 180,E1 33649.574,E2 33649.574} C_VEL
LIN {X 0,Y 15.587,Z 1240.5,A -85,B 0,C 180,E1 33649.574,E2 33649.574} C_VEL
LIN {X 0,Y 15.587,Z 1240.5,A -85,B 0,C 180,E1 33649.574,E2 33649.574}

